LIN {X 0,Y 236.728,Z 519.016,A -85,B 0,C 180,E1 -22919.006,E2 -22919.006} C_VEL
LIN {X 0,Y 244.263,Z 527.464,A -85,B 0,C 180,E1 -22920.717,E2 -22920.717} C_VEL
LIN {X 0,Y 253.073,Z 536.486,A -85,B 0,C 180,E1 -22922.703,E2 -22922.703} C_VEL
LIN {X 0,Y 263.693,Z 545.897,A -85,B 0,C 180,E1 -22924.98,E2 -22924.98} C_VEL
LIN {X 0,Y 276.829,Z 555.997,A -85,B 0,C 180,E1 -22927.616,E2 -22927.616} C_VEL
LIN {X 0,Y 290.969,Z 566.15,A -85,B 0,C 180,E1 -22930.387,E2 -22930.387} C_VEL
LIN {X 0,Y 300.035,Z 572.76,A -85,B 0,C 180,E1 -22932.271,E2 -22932.271} C_VEL
LIN {X 0,Y 305.154,Z 576.298,A -85,B 0,C 180,E1 -22933.437,E2 -22933.437} C_VEL
LIN {X 0,Y 312.329,Z 581.44,A -85,B 0,C 180,E1 -22935.368,E2 -22935.368} C_VEL
LIN {X 0,Y 318.737,Z 585.432,A -85,B 0,C 180,E1 -22937.262,E2 -22937.262} C_VEL
LIN {X 0,Y 322.774,Z 588.128,A -85,B 0,C 180,E1 -22938.699,E2 -22938.699} C_VEL
LIN {X 0,Y 327.517,Z 591.436,A -85,B 0,C 180,E1 -22940.777,E2 -22940.777} C_VEL
LIN {X 0,Y 331.257,Z 593.607,A -85,B 0,C 180,E1 -22942.686,E2 -22942.686} C_VEL
LIN {X 0,Y 333.425,Z 594.669,A -85,B 0,C 180,E1 -22943.95,E2 -22943.95} C_VEL
LIN {X 0,Y 335.159,Z 595.455,A -85,B 0,C 180,E1 -22945.188,E2 -22945.188} C_VEL
LIN {X 0,Y 336.581,Z 595.99,A -85,B 0,C 180,E1 -22946.408,E2 -22946.408} C_VEL
LIN {X 0,Y 337.614,Z 596.404,A -85,B 0,C 180,E1 -22947.687,E2 -22947.687} C_VEL
LIN {X 0,Y 338.056,Z 596.662,A -85,B 0,C 180,E1 -22948.808,E2 -22948.808} C_VEL
LIN {X 0,Y 338.329,Z 596.679,A -85,B 0,C 180,E1 -22950,E2 -22950} C_VEL
LIN {X 0,Y 338.087,Z 596.63,A -85,B 0,C 180,E1 -22951.191,E2 -22951.191} C_VEL
LIN {X 0,Y 337.557,Z 596.361,A -85,B 0,C 180,E1 -22952.386,E2 -22952.386} C_VEL
LIN {X 0,Y 336.568,Z 595.974,A -85,B 0,C 180,E1 -22953.591,E2 -22953.591} C_VEL
LIN {X 0,Y 335.099,Z 595.465,A -85,B 0,C 180,E1 -22954.812,E2 -22954.812} C_VEL
LIN {X 0,Y 332.514,Z 594.273,A -85,B 0,C 180,E1 -22956.599,E2 -22956.599} C_VEL
LIN {X 0,Y 327.516,Z 591.416,A -85,B 0,C 180,E1 -22959.222,E2 -22959.222} C_VEL
LIN {X 0,Y 322.595,Z 587.972,A -85,B 0,C 180,E1 -22961.378,E2 -22961.378} C_VEL
LIN {X 0,Y 317.51,Z 584.709,A -85,B 0,C 180,E1 -22963.116,E2 -22963.116} C_VEL
LIN {X 0,Y 312.34,Z 581.41,A -85,B 0,C 180,E1 -22964.64,E2 -22964.64} C_VEL
LIN {X 0,Y 305.088,Z 576.303,A -85,B 0,C 180,E1 -22966.566,E2 -22966.566} C_VEL
LIN {X 0,Y 298.32,Z 571.62,A -85,B 0,C 180,E1 -22968.091,E2 -22968.091} C_VEL
LIN {X 0,Y 288.226,Z 564.238,A -85,B 0,C 180,E1 -22970.155,E2 -22970.155} C_VEL
LIN {X 0,Y 274.506,Z 554.347,A -85,B 0,C 180,E1 -22972.829,E2 -22972.829} C_VEL
LIN {X 0,Y 261.578,Z 544.164,A -85,B 0,C 180,E1 -22975.459,E2 -22975.459} C_VEL
LIN {X 0,Y 249.228,Z 532.777,A -85,B 0,C 180,E1 -22978.145,E2 -22978.145} C_VEL
LIN {X 0,Y 238.85,Z 521.493,A -85,B 0,C 180,E1 -22980.508,E2 -22980.508} C_VEL
LIN {X 0,Y 230.342,Z 511.194,A -85,B 0,C 180,E1 -22982.456,E2 -22982.456} C_VEL
LIN {X 0,Y 222.039,Z 500.025,A -85,B 0,C 180,E1 -22984.323,E2 -22984.323} C_VEL
LIN {X 0,Y 214.349,Z 487.813,A -85,B 0,C 180,E1 -22986.246,E2 -22986.246} C_VEL
LIN {X 0,Y 207.911,Z 475.576,A -85,B 0,C 180,E1 -22988.093,E2 -22988.093} C_VEL
LIN {X 0,Y 200.375,Z 459.074,A -85,B 0,C 180,E1 -22990.575,E2 -22990.575} C_VEL
LIN {X 0,Y 193.887,Z 446.712,A -85,B 0,C 180,E1 -22992.86,E2 -22992.86} C_VEL
LIN {X 0,Y 186.703,Z 434.875,A -85,B 0,C 180,E1 -22995.592,E2 -22995.592} C_VEL
LIN {X 0,Y 180.616,Z 426.163,A -85,B 0,C 180,E1 -22998.122,E2 -22998.122} C_VEL
LIN {X 0,Y 177.895,Z 422.29,A -85,B 0,C 180,E1 -22999.351,E2 -22999.351} C_VEL
LIN {X 0,Y 175.543,Z 419.17,A -85,B 0,C 180,E1 -23000.457,E2 -23000.457} C_VEL
LIN {X 0,Y 174.806,Z 417.866,A -85,B 0,C 180,E1 -23000.836,E2 -23000.836} C_VEL
LIN {X 0,Y 172.532,Z 415.661,A -85,B 0,C 180,E1 -23001.925,E2 -23001.925} C_VEL
LIN {X 0,Y 171.492,Z 413.209,A -85,B 0,C 180,E1 -23002.718,E2 -23002.718} C_VEL
LIN {X 0,Y 171.419,Z 412.642,A -85,B 0,C 180,E1 -23003.526,E2 -23003.526} C_VEL
LIN {X 0,Y 171.453,Z 412.622,A -85,B 0,C 180,E1 -23009.405,E2 -23009.405} C_VEL
LIN {X 0,Y 171.464,Z 412.598,A -85,B 0,C 180,E1 -23014.384,E2 -23014.384} C_VEL
LIN {X 0,Y 171.575,Z 412.566,A -85,B 0,C 180,E1 -23020.873,E2 -23020.873} C_VEL
LIN {X 0,Y 171.606,Z 412.607,A -85,B 0,C 180,E1 -23025.777,E2 -23025.777} C_VEL
LIN {X 0,Y 171.887,Z 412.522,A -85,B 0,C 180,E1 -23030.588,E2 -23030.588} C_VEL
LIN {X 0,Y 171.822,Z 412.58,A -85,B 0,C 180,E1 -23035.309,E2 -23035.309} C_VEL
LIN {X 0,Y 172.328,Z 412.463,A -85,B 0,C 180,E1 -23040.001,E2 -23040.001} C_VEL
LIN {X 0,Y 171.822,Z 412.582,A -85,B 0,C 180,E1 -23044.694,E2 -23044.694} C_VEL
LIN {X 0,Y 171.871,Z 412.52,A -85,B 0,C 180,E1 -23049.415,E2 -23049.415} C_VEL
LIN {X 0,Y 171.601,Z 412.606,A -85,B 0,C 180,E1 -23054.226,E2 -23054.226} C_VEL
LIN {X 0,Y 171.542,Z 412.57,A -85,B 0,C 180,E1 -23059.563,E2 -23059.563} C_VEL
LIN {X 0,Y 171.461,Z 412.589,A -85,B 0,C 180,E1 -23065.613,E2 -23065.613} C_VEL
LIN {X 0,Y 171.457,Z 412.629,A -85,B 0,C 180,E1 -23070.598,E2 -23070.598} C_VEL
LIN {X 0,Y 171.435,Z 412.785,A -85,B 0,C 180,E1 -23076.473,E2 -23076.473} C_VEL
LIN {X 0,Y 171.688,Z 413.83,A -85,B 0,C 180,E1 -23077.143,E2 -23077.143} C_VEL
LIN {X 0,Y 173.195,Z 416.474,A -85,B 0,C 180,E1 -23078.023,E2 -23078.023} C_VEL
LIN {X 0,Y 175.673,Z 419.602,A -85,B 0,C 180,E1 -23079.236,E2 -23079.236} C_VEL
LIN {X 0,Y 178.708,Z 424.182,A -85,B 0,C 180,E1 -23080.681,E2 -23080.681} C_VEL
LIN {X 0,Y 184.514,Z 434.276,A -85,B 0,C 180,E1 -23083.285,E2 -23083.285} C_VEL
LIN {X 0,Y 191.758,Z 448.084,A -85,B 0,C 180,E1 -23086.225,E2 -23086.225} C_VEL
LIN {X 0,Y 198.367,Z 463.492,A -85,B 0,C 180,E1 -23088.744,E2 -23088.744} C_VEL
LIN {X 0,Y 200.007,Z 468.221,A -85,B 0,C 180,E1 -23089.371,E2 -23089.371} C_VEL
LIN {X 0,Y 201.452,Z 479.472,A -85,B 0,C 180,E1 -23090.232,E2 -23090.232} C_VEL
LIN {X 0,Y 199.102,Z 520.445,A -85,B 0,C 180,E1 -23091.619,E2 -23091.619} C_VEL
LIN {X 0,Y 198.002,Z 530.704,A -85,B 0,C 180,E1 -23092.185,E2 -23092.185} C_VEL
LIN {X 0,Y 196.533,Z 540.028,A -85,B 0,C 180,E1 -23092.884,E2 -23092.884} C_VEL
LIN {X 0,Y 194.673,Z 549.117,A -85,B 0,C 180,E1 -23093.762,E2 -23093.762} C_VEL
LIN {X 0,Y 192.446,Z 558.257,A -85,B 0,C 180,E1 -23094.889,E2 -23094.889} C_VEL
LIN {X 0,Y 189.964,Z 567.255,A -85,B 0,C 180,E1 -23096.294,E2 -23096.294} C_VEL
LIN {X 0,Y 187.186,Z 575.977,A -85,B 0,C 180,E1 -23097.973,E2 -23097.973} C_VEL
LIN {X 0,Y 184.617,Z 583.395,A -85,B 0,C 180,E1 -23099.71,E2 -23099.71} C_VEL
LIN {X 0,Y 181.224,Z 592.186,A -85,B 0,C 180,E1 -23102.267,E2 -23102.267} C_VEL
LIN {X 0,Y 178.889,Z 598.176,A -85,B 0,C 180,E1 -23104.397,E2 -23104.397} C_VEL
LIN {X 0,Y 176.422,Z 604.491,A -85,B 0,C 180,E1 -23107.146,E2 -23107.146} C_VEL
LIN {X 0,Y 174.145,Z 609.763,A -85,B 0,C 180,E1 -23109.939,E2 -23109.939} C_VEL
LIN {X 0,Y 171.876,Z 614.855,A -85,B 0,C 180,E1 -23113.369,E2 -23113.369} C_VEL
LIN {X 0,Y 170.402,Z 618.826,A -85,B 0,C 180,E1 -23116.89,E2 -23116.89} C_VEL
LIN {X 0,Y 169.425,Z 621.766,A -85,B 0,C 180,E1 -23120.45,E2 -23120.45} C_VEL
LIN {X 0,Y 169.076,Z 623.272,A -85,B 0,C 180,E1 -23122.837,E2 -23122.837} C_VEL
LIN {X 0,Y 168.87,Z 624.806,A -85,B 0,C 180,E1 -23127.616,E2 -23127.616} C_VEL
LIN {X 0,Y 168.968,Z 625.09,A -85,B 0,C 180,E1 -23130.001,E2 -23130.001} C_VEL
LIN {X 0,Y 168.866,Z 624.204,A -85,B 0,C 180,E1 -23134.775,E2 -23134.775} C_VEL
LIN {X 0,Y 169.043,Z 623.271,A -85,B 0,C 180,E1 -23137.166,E2 -23137.166} C_VEL
LIN {X 0,Y 169.229,Z 622.38,A -85,B 0,C 180,E1 -23138.579,E2 -23138.579} C_VEL
LIN {X 0,Y 168.959,Z 621.139,A -85,B 0,C 180,E1 -23140.532,E2 -23140.532} C_VEL
LIN {X 0,Y 167.045,Z 618.534,A -85,B 0,C 180,E1 -23143.742,E2 -23143.742} C_VEL
LIN {X 0,Y 165.569,Z 615.248,A -85,B 0,C 180,E1 -23146.93,E2 -23146.93} C_VEL
LIN {X 0,Y 165.975,Z 612.775,A -85,B 0,C 180,E1 -23148.781,E2 -23148.781} C_VEL
LIN {X 0,Y 168.814,Z 606.475,A -85,B 0,C 180,E1 -23152.65,E2 -23152.65} C_VEL
LIN {X 0,Y 171.166,Z 601.299,A -85,B 0,C 180,E1 -23155.195,E2 -23155.195} C_VEL
LIN {X 0,Y 173.701,Z 595.108,A -85,B 0,C 180,E1 -23157.73,E2 -23157.73} C_VEL
LIN {X 0,Y 177.091,Z 586.895,A -85,B 0,C 180,E1 -23160.398,E2 -23160.398} C_VEL
LIN {X 0,Y 180.045,Z 579.071,A -85,B 0,C 180,E1 -23162.461,E2 -23162.461} C_VEL
LIN {X 0,Y 182.872,Z 570.992,A -85,B 0,C 180,E1 -23164.198,E2 -23164.198} C_VEL
LIN {X 0,Y 185.848,Z 561.234,A -85,B 0,C 180,E1 -23165.884,E2 -23165.884} C_VEL
LIN {X 0,Y 188.042,Z 552.846,A -85,B 0,C 180,E1 -23167.061,E2 -23167.061} C_VEL
LIN {X 0,Y 190.44,Z 542.345,A -85,B 0,C 180,E1 -23168.181,E2 -23168.181} C_VEL
LIN {X 0,Y 192.255,Z 532.052,A -85,B 0,C 180,E1 -23169.006,E2 -23169.006} C_VEL
LIN {X 0,Y 193.52,Z 521.679,A -85,B 0,C 180,E1 -23169.604,E2 -23169.604} C_VEL
LIN {X 0,Y 194.902,Z 499.84,A -85,B 0,C 180,E1 -23170.408,E2 -23170.408} C_VEL
LIN {X 0,Y 196.016,Z 479.708,A -85,B 0,C 180,E1 -23171.083,E2 -23171.083} C_VEL
LIN {X 0,Y 194.546,Z 469.953,A -85,B 0,C 180,E1 -23171.929,E2 -23171.929} C_VEL
LIN {X 0,Y 189.397,Z 457.055,A -85,B 0,C 180,E1 -23173.995,E2 -23173.995} C_VEL
LIN {X 0,Y 184.711,Z 447.009,A -85,B 0,C 180,E1 -23175.951,E2 -23175.951} C_VEL
LIN {X 0,Y 177.652,Z 433.788,A -85,B 0,C 180,E1 -23179.132,E2 -23179.132} C_VEL
LIN {X 0,Y 174.281,Z 428.326,A -85,B 0,C 180,E1 -23180.766,E2 -23180.766} C_VEL
LIN {X 0,Y 171.198,Z 423.48,A -85,B 0,C 180,E1 -23182.362,E2 -23182.362} C_VEL
LIN {X 0,Y 168.739,Z 420.14,A -85,B 0,C 180,E1 -23183.684,E2 -23183.684} C_VEL
LIN {X 0,Y 167.958,Z 418.839,A -85,B 0,C 180,E1 -23184.138,E2 -23184.138} C_VEL
LIN {X 0,Y 165.556,Z 416.617,A -85,B 0,C 180,E1 -23185.461,E2 -23185.461} C_VEL
LIN {X 0,Y 164.44,Z 414.112,A -85,B 0,C 180,E1 -23186.42,E2 -23186.42} C_VEL
LIN {X 0,Y 164.376,Z 413.526,A -85,B 0,C 180,E1 -23187.273,E2 -23187.273} C_VEL
LIN {X 0,Y 164.343,Z 413.477,A -85,B 0,C 180,E1 -23191.938,E2 -23191.938} C_VEL
LIN {X 0,Y 164.413,Z 413.469,A -85,B 0,C 180,E1 -23194.692,E2 -23194.692} C_VEL
LIN {X 0,Y 164.487,Z 413.451,A -85,B 0,C 180,E1 -23200.05,E2 -23200.05} C_VEL
LIN {X 0,Y 164.546,Z 413.477,A -85,B 0,C 180,E1 -23205.15,E2 -23205.15} C_VEL
LIN {X 0,Y 164.799,Z 413.4,A -85,B 0,C 180,E1 -23210.177,E2 -23210.177} C_VEL
LIN {X 0,Y 164.848,Z 413.407,A -85,B 0,C 180,E1 -23212.65,E2 -23212.65} C_VEL
LIN {X 0,Y 165.051,Z 413.393,A -85,B 0,C 180,E1 -23217.558,E2 -23217.558} C_VEL
LIN {X 0,Y 165.294,Z 413.339,A -85,B 0,C 180,E1 -23219.999,E2 -23219.999} C_VEL
LIN {X 0,Y 164.775,Z 413.459,A -85,B 0,C 180,E1 -23224.892,E2 -23224.892} C_VEL
LIN {X 0,Y 164.855,Z 413.419,A -85,B 0,C 180,E1 -23227.347,E2 -23227.347} C_VEL
LIN {X 0,Y 164.745,Z 413.413,A -85,B 0,C 180,E1 -23231.134,E2 -23231.134} C_VEL
LIN {X 0,Y 164.504,Z 413.456,A -85,B 0,C 180,E1 -23237.399,E2 -23237.399} C_VEL
LIN {X 0,Y 164.473,Z 413.451,A -85,B 0,C 180,E1 -23239.988,E2 -23239.988} C_VEL
LIN {X 0,Y 164.387,Z 413.474,A -85,B 0,C 180,E1 -23246.128,E2 -23246.128} C_VEL
LIN {X 0,Y 164.385,Z 413.492,A -85,B 0,C 180,E1 -23252.376,E2 -23252.376} C_VEL
LIN {X 0,Y 164.377,Z 413.826,A -85,B 0,C 180,E1 -23253.765,E2 -23253.765} C_VEL
LIN {X 0,Y 164.719,Z 415.071,A -85,B 0,C 180,E1 -23254.363,E2 -23254.363} C_VEL
LIN {X 0,Y 166.421,Z 417.681,A -85,B 0,C 180,E1 -23255.43,E2 -23255.43} C_VEL
LIN {X 0,Y 168.282,Z 419.225,A -85,B 0,C 180,E1 -23256.427,E2 -23256.427} C_VEL
LIN {X 0,Y 170.447,Z 422.668,A -85,B 0,C 180,E1 -23257.643,E2 -23257.643} C_VEL
LIN {X 0,Y 172.045,Z 424.419,A -85,B 0,C 180,E1 -23258.448,E2 -23258.448} C_VEL
LIN {X 0,Y 174.727,Z 428.084,A -85,B 0,C 180,E1 -23259.782,E2 -23259.782} C_VEL
LIN {X 0,Y 181.199,Z 437.59,A -85,B 0,C 180,E1 -23262.745,E2 -23262.745} C_VEL
LIN {X 0,Y 186.924,Z 446.683,A -85,B 0,C 180,E1 -23265.11,E2 -23265.11} C_VEL
LIN {X 0,Y 192.646,Z 456.992,A -85,B 0,C 180,E1 -23267.308,E2 -23267.308} C_VEL
LIN {X 0,Y 199.199,Z 470.707,A -85,B 0,C 180,E1 -23269.675,E2 -23269.675} C_VEL
LIN {X 0,Y 206.608,Z 486.849,A -85,B 0,C 180,E1 -23272.111,E2 -23272.111} C_VEL
LIN {X 0,Y 215.246,Z 501.527,A -85,B 0,C 180,E1 -23274.484,E2 -23274.484} C_VEL
LIN {X 0,Y 223.669,Z 513.611,A -85,B 0,C 180,E1 -23276.575,E2 -23276.575} C_VEL
LIN {X 0,Y 233.428,Z 525.815,A -85,B 0,C 180,E1 -23279.036,E2 -23279.036} C_VEL
LIN {X 0,Y 242.728,Z 536.201,A -85,B 0,C 180,E1 -23281.369,E2 -23281.369} C_VEL
LIN {X 0,Y 253.999,Z 546.99,A -85,B 0,C 180,E1 -23284.058,E2 -23284.058} C_VEL
LIN {X 0,Y 267.274,Z 557.559,A -85,B 0,C 180,E1 -23286.971,E2 -23286.971} C_VEL
LIN {X 0,Y 280.838,Z 567.195,A -85,B 0,C 180,E1 -23289.787,E2 -23289.787} C_VEL
LIN {X 0,Y 289.684,Z 573.411,A -85,B 0,C 180,E1 -23291.615,E2 -23291.615} C_VEL
LIN {X 0,Y 298.819,Z 579.758,A -85,B 0,C 180,E1 -23293.606,E2 -23293.606} C_VEL
LIN {X 0,Y 305.423,Z 584.503,A -85,B 0,C 180,E1 -23295.338,E2 -23295.338} C_VEL
LIN {X 0,Y 311.033,Z 588.132,A -85,B 0,C 180,E1 -23296.941,E2 -23296.941} C_VEL
LIN {X 0,Y 315.717,Z 591.005,A -85,B 0,C 180,E1 -23298.443,E2 -23298.443} C_VEL
LIN {X 0,Y 320.624,Z 594.537,A -85,B 0,C 180,E1 -23300.53,E2 -23300.53} C_VEL
LIN {X 0,Y 324.704,Z 597.007,A -85,B 0,C 180,E1 -23302.538,E2 -23302.538} C_VEL
LIN {X 0,Y 327,Z 598.172,A -85,B 0,C 180,E1 -23303.831,E2 -23303.831} C_VEL
LIN {X 0,Y 328.877,Z 599.073,A -85,B 0,C 180,E1 -23305.096,E2 -23305.096} C_VEL
LIN {X 0,Y 330.825,Z 599.849,A -85,B 0,C 180,E1 -23306.805,E2 -23306.805} C_VEL
LIN {X 0,Y 331.432,Z 600.068,A -85,B 0,C 180,E1 -23307.569,E2 -23307.569} C_VEL
LIN {X 0,Y 331.976,Z 600.353,A -85,B 0,C 180,E1 -23308.787,E2 -23308.787} C_VEL
LIN {X 0,Y 332.28,Z 600.374,A -85,B 0,C 180,E1 -23310,E2 -23310} C_VEL
LIN {X 0,Y 332.008,Z 600.326,A -85,B 0,C 180,E1 -23311.213,E2 -23311.213} C_VEL
LIN {X 0,Y 330.825,Z 599.859,A -85,B 0,C 180,E1 -23313.194,E2 -23313.194} C_VEL
LIN {X 0,Y 328.815,Z 599.085,A -85,B 0,C 180,E1 -23314.904,E2 -23314.904} C_VEL
LIN {X 0,Y 325.669,Z 597.531,A -85,B 0,C 180,E1 -23316.939,E2 -23316.939} C_VEL
LIN {X 0,Y 322.095,Z 595.476,A -85,B 0,C 180,E1 -23318.785,E2 -23318.785} C_VEL
LIN {X 0,Y 319.133,Z 593.487,A -85,B 0,C 180,E1 -23320.147,E2 -23320.147} C_VEL
LIN {X 0,Y 315.653,Z 590.975,A -85,B 0,C 180,E1 -23321.581,E2 -23321.581} C_VEL
LIN {X 0,Y 310.442,Z 587.771,A -85,B 0,C 180,E1 -23323.233,E2 -23323.233} C_VEL
LIN {X 0,Y 305.203,Z 584.349,A -85,B 0,C 180,E1 -23324.731,E2 -23324.731} C_VEL
LIN {X 0,Y 298.782,Z 579.747,A -85,B 0,C 180,E1 -23326.395,E2 -23326.395} C_VEL
LIN {X 0,Y 289.661,Z 573.417,A -85,B 0,C 180,E1 -23328.385,E2 -23328.385} C_VEL
LIN {X 0,Y 278.12,Z 565.341,A -85,B 0,C 180,E1 -23330.778,E2 -23330.778} C_VEL
LIN {X 0,Y 263.246,Z 554.562,A -85,B 0,C 180,E1 -23333.883,E2 -23333.883} C_VEL
LIN {X 0,Y 251.277,Z 544.483,A -85,B 0,C 180,E1 -23336.583,E2 -23336.583} C_VEL
LIN {X 0,Y 241.139,Z 534.456,A -85,B 0,C 180,E1 -23339.034,E2 -23339.034} C_VEL
LIN {X 0,Y 231.156,Z 523.114,A -85,B 0,C 180,E1 -23341.534,E2 -23341.534} C_VEL
LIN {X 0,Y 222.069,Z 511.424,A -85,B 0,C 180,E1 -23343.826,E2 -23343.826} C_VEL
LIN {X 0,Y 212.518,Z 497.302,A -85,B 0,C 180,E1 -23346.22,E2 -23346.22} C_VEL
LIN {X 0,Y 204.497,Z 482.639,A -85,B 0,C 180,E1 -23348.54,E2 -23348.54} C_VEL
LIN {X 0,Y 195.455,Z 462.655,A -85,B 0,C 180,E1 -23351.657,E2 -23351.657} C_VEL
LIN {X 0,Y 189.424,Z 450.986,A -85,B 0,C 180,E1 -23353.914,E2 -23353.914} C_VEL
LIN {X 0,Y 182.648,Z 439.754,A -85,B 0,C 180,E1 -23356.64,E2 -23356.64} C_VEL
LIN {X 0,Y 177.085,Z 431.544,A -85,B 0,C 180,E1 -23359.093,E2 -23359.093} C_VEL
LIN {X 0,Y 174.236,Z 427.557,A -85,B 0,C 180,E1 -23360.447,E2 -23360.447} C_VEL
LIN {X 0,Y 171.306,Z 423.48,A -85,B 0,C 180,E1 -23361.929,E2 -23361.929} C_VEL
LIN {X 0,Y 169.048,Z 420.726,A -85,B 0,C 180,E1 -23363.116,E2 -23363.116} C_VEL
LIN {X 0,Y 167.933,Z 418.825,A -85,B 0,C 180,E1 -23363.764,E2 -23363.764} C_VEL
LIN {X 0,Y 165.584,Z 416.669,A -85,B 0,C 180,E1 -23365.057,E2 -23365.057} C_VEL
LIN {X 0,Y 164.44,Z 414.038,A -85,B 0,C 180,E1 -23366.041,E2 -23366.041} C_VEL
LIN {X 0,Y 164.345,Z 413.513,A -85,B 0,C 180,E1 -23366.923,E2 -23366.923} C_VEL
LIN {X 0,Y 164.401,Z 413.504,A -85,B 0,C 180,E1 -23369.138,E2 -23369.138} C_VEL
LIN {X 0,Y 164.412,Z 413.479,A -85,B 0,C 180,E1 -23374.695,E2 -23374.695} C_VEL
LIN {X 0,Y 164.48,Z 413.45,A -85,B 0,C 180,E1 -23380.052,E2 -23380.052} C_VEL
LIN {X 0,Y 164.549,Z 413.489,A -85,B 0,C 180,E1 -23385.153,E2 -23385.153} C_VEL
LIN {X 0,Y 164.801,Z 413.402,A -85,B 0,C 180,E1 -23390.18,E2 -23390.18} C_VEL
LIN {X 0,Y 164.851,Z 413.419,A -85,B 0,C 180,E1 -23392.653,E2 -23392.653} C_VEL
LIN {X 0,Y 165.047,Z 413.382,A -85,B 0,C 180,E1 -23397.561,E2 -23397.561} C_VEL
LIN {X 0,Y 165.291,Z 413.339,A -85,B 0,C 180,E1 -23400.001,E2 -23400.001} C_VEL
LIN {X 0,Y 164.771,Z 413.46,A -85,B 0,C 180,E1 -23404.895,E2 -23404.895} C_VEL
LIN {X 0,Y 164.844,Z 413.408,A -85,B 0,C 180,E1 -23407.35,E2 -23407.35} C_VEL
LIN {X 0,Y 164.748,Z 413.416,A -85,B 0,C 180,E1 -23411.148,E2 -23411.148} C_VEL
LIN {X 0,Y 164.49,Z 413.447,A -85,B 0,C 180,E1 -23417.404,E2 -23417.404} C_VEL
LIN {X 0,Y 164.472,Z 413.453,A -85,B 0,C 180,E1 -23419.991,E2 -23419.991} C_VEL
LIN {X 0,Y 164.387,Z 413.467,A -85,B 0,C 180,E1 -23426.132,E2 -23426.132} C_VEL
LIN {X 0,Y 164.388,Z 413.505,A -85,B 0,C 180,E1 -23432.38,E2 -23432.38} C_VEL
LIN {X 0,Y 164.388,Z 413.886,A -85,B 0,C 180,E1 -23433.418,E2 -23433.418} C_VEL
LIN {X 0,Y 164.851,Z 415.357,A -85,B 0,C 180,E1 -23434.077,E2 -23434.077} C_VEL
LIN {X 0,Y 166.518,Z 417.759,A -85,B 0,C 180,E1 -23435.097,E2 -23435.097} C_VEL
LIN {X 0,Y 168.305,Z 419.258,A -85,B 0,C 180,E1 -23436.054,E2 -23436.054} C_VEL
LIN {X 0,Y 170.355,Z 422.505,A -85,B 0,C 180,E1 -23437.205,E2 -23437.205} C_VEL
LIN {X 0,Y 172.352,Z 425.179,A -85,B 0,C 180,E1 -23438.241,E2 -23438.241} C_VEL
LIN {X 0,Y 176.255,Z 431.544,A -85,B 0,C 180,E1 -23440.206,E2 -23440.206} C_VEL
LIN {X 0,Y 180.512,Z 439.006,A -85,B 0,C 180,E1 -23442.202,E2 -23442.202} C_VEL
LIN {X 0,Y 187.332,Z 452.339,A -85,B 0,C 180,E1 -23445.148,E2 -23445.148} C_VEL
LIN {X 0,Y 194.157,Z 468.716,A -85,B 0,C 180,E1 -23447.908,E2 -23447.908} C_VEL
LIN {X 0,Y 194.9,Z 471.646,A -85,B 0,C 180,E1 -23448.245,E2 -23448.245} C_VEL
LIN {X 0,Y 195.961,Z 480.953,A -85,B 0,C 180,E1 -23448.963,E2 -23448.963} C_VEL
LIN {X 0,Y 193.606,Z 520.134,A -85,B 0,C 180,E1 -23450.311,E2 -23450.311} C_VEL
LIN {X 0,Y 192.382,Z 530.958,A -85,B 0,C 180,E1 -23450.918,E2 -23450.918} C_VEL
LIN {X 0,Y 190.676,Z 541.095,A -85,B 0,C 180,E1 -23451.709,E2 -23451.709} C_VEL
LIN {X 0,Y 188.532,Z 550.889,A -85,B 0,C 180,E1 -23452.718,E2 -23452.718} C_VEL
LIN {X 0,Y 186.248,Z 559.651,A -85,B 0,C 180,E1 -23453.873,E2 -23453.873} C_VEL
LIN {X 0,Y 183.674,Z 568.372,A -85,B 0,C 180,E1 -23455.309,E2 -23455.309} C_VEL
LIN {X 0,Y 180.799,Z 576.879,A -85,B 0,C 180,E1 -23457.031,E2 -23457.031} C_VEL
LIN {X 0,Y 178.49,Z 583.199,A -85,B 0,C 180,E1 -23458.554,E2 -23458.554} C_VEL
LIN {X 0,Y 174.946,Z 591.99,A -85,B 0,C 180,E1 -23461.181,E2 -23461.181} C_VEL
LIN {X 0,Y 172.483,Z 597.98,A -85,B 0,C 180,E1 -23463.372,E2 -23463.372} C_VEL
LIN {X 0,Y 169.872,Z 604.295,A -85,B 0,C 180,E1 -23466.211,E2 -23466.211} C_VEL
LIN {X 0,Y 167.452,Z 609.567,A -85,B 0,C 180,E1 -23469.1,E2 -23469.1} C_VEL
LIN {X 0,Y 165.068,Z 614.66,A -85,B 0,C 180,E1 -23472.661,E2 -23472.661} C_VEL
LIN {X 0,Y 163.452,Z 618.629,A -85,B 0,C 180,E1 -23476.322,E2 -23476.322} C_VEL
LIN {X 0,Y 162.405,Z 621.571,A -85,B 0,C 180,E1 -23480.033,E2 -23480.033} C_VEL
LIN {X 0,Y 162.002,Z 623.076,A -85,B 0,C 180,E1 -23482.523,E2 -23482.523} C_VEL
LIN {X 0,Y 161.8,Z 624.612,A -85,B 0,C 180,E1 -23487.511,E2 -23487.511} C_VEL
LIN {X 0,Y 161.884,Z 624.895,A -85,B 0,C 180,E1 -23490.001,E2 -23490.001} C_VEL
LIN {X 0,Y 161.771,Z 624.009,A -85,B 0,C 180,E1 -23494.985,E2 -23494.985} C_VEL
LIN {X 0,Y 162.149,Z 622.327,A -85,B 0,C 180,E1 -23498.719,E2 -23498.719} C_VEL
LIN {X 0,Y 163.452,Z 618.628,A -85,B 0,C 180,E1 -23503.68,E2 -23503.68} C_VEL
LIN {X 0,Y 165.063,Z 614.658,A -85,B 0,C 180,E1 -23507.341,E2 -23507.341} C_VEL
LIN {X 0,Y 165.975,Z 612.775,A -85,B 0,C 180,E1 -23508.781,E2 -23508.781} C_VEL
LIN {X 0,Y 166.522,Z 610.192,A -85,B 0,C 180,E1 -23510.581,E2 -23510.581} C_VEL
LIN {X 0,Y 165.941,Z 605.51,A -85,B 0,C 180,E1 -23513.589,E2 -23513.589} C_VEL
LIN {X 0,Y 165.656,Z 600.32,A -85,B 0,C 180,E1 -23516.524,E2 -23516.524} C_VEL
LIN {X 0,Y 166.652,Z 596.784,A -85,B 0,C 180,E1 -23518.148,E2 -23518.148} C_VEL
LIN {X 0,Y 170.23,Z 588.548,A -85,B 0,C 180,E1 -23521.069,E2 -23521.069} C_VEL
LIN {X 0,Y 174.084,Z 578.875,A -85,B 0,C 180,E1 -23523.718,E2 -23523.718} C_VEL
LIN {X 0,Y 177.046,Z 570.797,A -85,B 0,C 180,E1 -23525.49,E2 -23525.49} C_VEL
LIN {X 0,Y 180.134,Z 561.039,A -85,B 0,C 180,E1 -23527.21,E2 -23527.21} C_VEL
LIN {X 0,Y 182.441,Z 552.651,A -85,B 0,C 180,E1 -23528.402,E2 -23528.402} C_VEL
LIN {X 0,Y 184.919,Z 542.151,A -85,B 0,C 180,E1 -23529.539,E2 -23529.539} C_VEL
LIN {X 0,Y 186.827,Z 531.734,A -85,B 0,C 180,E1 -23530.38,E2 -23530.38} C_VEL
LIN {X 0,Y 188.082,Z 521.544,A -85,B 0,C 180,E1 -23530.985,E2 -23530.985} C_VEL
LIN {X 0,Y 189.541,Z 499.766,A -85,B 0,C 180,E1 -23531.797,E2 -23531.797} C_VEL
LIN {X 0,Y 190.654,Z 480.823,A -85,B 0,C 180,E1 -23532.437,E2 -23532.437} C_VEL
LIN {X 0,Y 189.402,Z 472.537,A -85,B 0,C 180,E1 -23533.202,E2 -23533.202} C_VEL
LIN {X 0,Y 184.087,Z 459.259,A -85,B 0,C 180,E1 -23535.482,E2 -23535.482} C_VEL
LIN {X 0,Y 180.111,Z 450.731,A -85,B 0,C 180,E1 -23537.261,E2 -23537.261} C_VEL
LIN {X 0,Y 173.86,Z 438.725,A -85,B 0,C 180,E1 -23540.275,E2 -23540.275} C_VEL
LIN {X 0,Y 170.411,Z 432.987,A -85,B 0,C 180,E1 -23542.064,E2 -23542.064} C_VEL
LIN {X 0,Y 167.99,Z 429.046,A -85,B 0,C 180,E1 -23543.403,E2 -23543.403} C_VEL
LIN {X 0,Y 165.336,Z 425.183,A -85,B 0,C 180,E1 -23544.935,E2 -23544.935} C_VEL
LIN {X 0,Y 162.486,Z 422.107,A -85,B 0,C 180,E1 -23546.623,E2 -23546.623} C_VEL
LIN {X 0,Y 161.16,Z 419.831,A -85,B 0,C 180,E1 -23547.523,E2 -23547.523} C_VEL
LIN {X 0,Y 158.833,Z 417.904,A -85,B 0,C 180,E1 -23549.021,E2 -23549.021} C_VEL
LIN {X 0,Y 157.408,Z 414.944,A -85,B 0,C 180,E1 -23550.4,E2 -23550.4} C_VEL
LIN {X 0,Y 157.299,Z 414.413,A -85,B 0,C 180,E1 -23551.294,E2 -23551.294} C_VEL
LIN {X 0,Y 157.313,Z 414.373,A -85,B 0,C 180,E1 -23556.29,E2 -23556.29} C_VEL
LIN {X 0,Y 157.417,Z 414.324,A -85,B 0,C 180,E1 -23561.787,E2 -23561.787} C_VEL
LIN {X 0,Y 157.552,Z 414.338,A -85,B 0,C 180,E1 -23567.111,E2 -23567.111} C_VEL
LIN {X 0,Y 157.728,Z 414.282,A -85,B 0,C 180,E1 -23569.732,E2 -23569.732} C_VEL
LIN {X 0,Y 157.805,Z 414.279,A -85,B 0,C 180,E1 -23572.32,E2 -23572.32} C_VEL
LIN {X 0,Y 158.257,Z 414.214,A -85,B 0,C 180,E1 -23579.999,E2 -23579.999} C_VEL
LIN {X 0,Y 157.811,Z 414.289,A -85,B 0,C 180,E1 -23587.676,E2 -23587.676} C_VEL
LIN {X 0,Y 157.676,Z 414.293,A -85,B 0,C 180,E1 -23591.306,E2 -23591.306} C_VEL
LIN {X 0,Y 157.478,Z 414.36,A -85,B 0,C 180,E1 -23595.53,E2 -23595.53} C_VEL
LIN {X 0,Y 157.369,Z 414.342,A -85,B 0,C 180,E1 -23600.931,E2 -23600.931} C_VEL
LIN {X 0,Y 157.308,Z 414.351,A -85,B 0,C 180,E1 -23606.679,E2 -23606.679} C_VEL
LIN {X 0,Y 157.339,Z 414.676,A -85,B 0,C 180,E1 -23609.703,E2 -23609.703} C_VEL
LIN {X 0,Y 157.689,Z 415.857,A -85,B 0,C 180,E1 -23610.46,E2 -23610.46} C_VEL
LIN {X 0,Y 159.215,Z 418.377,A -85,B 0,C 180,E1 -23611.632,E2 -23611.632} C_VEL
LIN {X 0,Y 161.46,Z 420.154,A -85,B 0,C 180,E1 -23613.054,E2 -23613.054} C_VEL
LIN {X 0,Y 163.49,Z 423.459,A -85,B 0,C 180,E1 -23614.394,E2 -23614.394} C_VEL
LIN {X 0,Y 165.522,Z 425.569,A -85,B 0,C 180,E1 -23615.571,E2 -23615.571} C_VEL
LIN {X 0,Y 167.969,Z 429.04,A -85,B 0,C 180,E1 -23616.973,E2 -23616.973} C_VEL
LIN {X 0,Y 169.204,Z 430.642,A -85,B 0,C 180,E1 -23617.639,E2 -23617.639} C_VEL
LIN {X 0,Y 175.22,Z 439.293,A -85,B 0,C 180,E1 -23620.675,E2 -23620.675} C_VEL
LIN {X 0,Y 181.544,Z 449.222,A -85,B 0,C 180,E1 -23623.524,E2 -23623.524} C_VEL
LIN {X 0,Y 187.875,Z 460.689,A -85,B 0,C 180,E1 -23626.135,E2 -23626.135} C_VEL
LIN {X 0,Y 193.898,Z 473.486,A -85,B 0,C 180,E1 -23628.458,E2 -23628.458} C_VEL
LIN {X 0,Y 201.993,Z 491.356,A -85,B 0,C 180,E1 -23631.279,E2 -23631.279} C_VEL
LIN {X 0,Y 210.523,Z 506.075,A -85,B 0,C 180,E1 -23633.746,E2 -23633.746} C_VEL
LIN {X 0,Y 218.434,Z 517.873,A -85,B 0,C 180,E1 -23635.942,E2 -23635.942} C_VEL
LIN {X 0,Y 227.023,Z 529.009,A -85,B 0,C 180,E1 -23638.352,E2 -23638.352} C_VEL
LIN {X 0,Y 234.425,Z 537.612,A -85,B 0,C 180,E1 -23640.388,E2 -23640.388} C_VEL
LIN {X 0,Y 244.429,Z 547.815,A -85,B 0,C 180,E1 -23643.039,E2 -23643.039} C_VEL
LIN {X 0,Y 254.755,Z 556.641,A -85,B 0,C 180,E1 -23645.555,E2 -23645.555} C_VEL
LIN {X 0,Y 269.098,Z 567.114,A -85,B 0,C 180,E1 -23648.778,E2 -23648.778} C_VEL
LIN {X 0,Y 281.65,Z 575.581,A -85,B 0,C 180,E1 -23651.477,E2 -23651.477} C_VEL
LIN {X 0,Y 292.579,Z 582.992,A -85,B 0,C 180,E1 -23653.908,E2 -23653.908} C_VEL
LIN {X 0,Y 299.527,Z 587.974,A -85,B 0,C 180,E1 -23655.705,E2 -23655.705} C_VEL
LIN {X 0,Y 304.737,Z 591.358,A -85,B 0,C 180,E1 -23657.167,E2 -23657.167} C_VEL
LIN {X 0,Y 309.786,Z 594.475,A -85,B 0,C 180,E1 -23658.77,E2 -23658.77} C_VEL
LIN {X 0,Y 315.026,Z 598.177,A -85,B 0,C 180,E1 -23661.015,E2 -23661.015} C_VEL
LIN {X 0,Y 318.736,Z 600.427,A -85,B 0,C 180,E1 -23662.847,E2 -23662.847} C_VEL
LIN {X 0,Y 322.233,Z 602.162,A -85,B 0,C 180,E1 -23664.995,E2 -23664.995} C_VEL
LIN {X 0,Y 323.946,Z 602.89,A -85,B 0,C 180,E1 -23666.334,E2 -23666.334} C_VEL
LIN {X 0,Y 325.059,Z 603.308,A -85,B 0,C 180,E1 -23667.521,E2 -23667.521} C_VEL
LIN {X 0,Y 325.655,Z 603.606,A -85,B 0,C 180,E1 -23668.763,E2 -23668.763} C_VEL
LIN {X 0,Y 325.97,Z 603.643,A -85,B 0,C 180,E1 -23670,E2 -23670} C_VEL
LIN {X 0,Y 325.678,Z 603.588,A -85,B 0,C 180,E1 -23671.236,E2 -23671.236} C_VEL
LIN {X 0,Y 325.059,Z 603.298,A -85,B 0,C 180,E1 -23672.478,E2 -23672.478} C_VEL
LIN {X 0,Y 323.85,Z 602.851,A -85,B 0,C 180,E1 -23673.732,E2 -23673.732} C_VEL
LIN {X 0,Y 322.2,Z 602.171,A -85,B 0,C 180,E1 -23675.005,E2 -23675.005} C_VEL
LIN {X 0,Y 320.222,Z 601.202,A -85,B 0,C 180,E1 -23676.3,E2 -23676.3} C_VEL
LIN {X 0,Y 317.783,Z 599.904,A -85,B 0,C 180,E1 -23677.625,E2 -23677.625} C_VEL
LIN {X 0,Y 313.631,Z 597.242,A -85,B 0,C 180,E1 -23679.613,E2 -23679.613} C_VEL
LIN {X 0,Y 309.784,Z 594.458,A -85,B 0,C 180,E1 -23681.229,E2 -23681.229} C_VEL
LIN {X 0,Y 304.734,Z 591.384,A -85,B 0,C 180,E1 -23682.83,E2 -23682.83} C_VEL
LIN {X 0,Y 297.951,Z 586.837,A -85,B 0,C 180,E1 -23684.742,E2 -23684.742} C_VEL
LIN {X 0,Y 292.574,Z 583.008,A -85,B 0,C 180,E1 -23686.088,E2 -23686.088} C_VEL
LIN {X 0,Y 281.641,Z 575.61,A -85,B 0,C 180,E1 -23688.518,E2 -23688.518} C_VEL
LIN {X 0,Y 267.45,Z 565.985,A -85,B 0,C 180,E1 -23691.585,E2 -23691.585} C_VEL
LIN {X 0,Y 253.442,Z 555.619,A -85,B 0,C 180,E1 -23694.75,E2 -23694.75} C_VEL
LIN {X 0,Y 241.263,Z 544.795,A -85,B 0,C 180,E1 -23697.779,E2 -23697.779} C_VEL
LIN {X 0,Y 230.745,Z 533.491,A -85,B 0,C 180,E1 -23700.613,E2 -23700.613} C_VEL
LIN {X 0,Y 221.966,Z 522.576,A -85,B 0,C 180,E1 -23703.066,E2 -23703.066} C_VEL
LIN {X 0,Y 214.582,Z 512.309,A -85,B 0,C 180,E1 -23705.139,E2 -23705.139} C_VEL
LIN {X 0,Y 205.92,Z 498.513,A -85,B 0,C 180,E1 -23707.534,E2 -23707.534} C_VEL
LIN {X 0,Y 199.124,Z 485.472,A -85,B 0,C 180,E1 -23709.66,E2 -23709.66} C_VEL
LIN {X 0,Y 190.831,Z 466.717,A -85,B 0,C 180,E1 -23712.709,E2 -23712.709} C_VEL
LIN {X 0,Y 184.918,Z 455.087,A -85,B 0,C 180,E1 -23715.061,E2 -23715.061} C_VEL
LIN {X 0,Y 178.882,Z 444.895,A -85,B 0,C 180,E1 -23717.64,E2 -23717.64} C_VEL
LIN {X 0,Y 173.249,Z 436.424,A -85,B 0,C 180,E1 -23720.277,E2 -23720.277} C_VEL
LIN {X 0,Y 170.439,Z 432.474,A -85,B 0,C 180,E1 -23721.7,E2 -23721.7} C_VEL
LIN {X 0,Y 168.09,Z 429.142,A -85,B 0,C 180,E1 -23722.964,E2 -23722.964} C_VEL
LIN {X 0,Y 165.523,Z 425.593,A -85,B 0,C 180,E1 -23724.427,E2 -23724.427} C_VEL
LIN {X 0,Y 162.258,Z 421.734,A -85,B 0,C 180,E1 -23726.387,E2 -23726.387} C_VEL
LIN {X 0,Y 161.136,Z 419.835,A -85,B 0,C 180,E1 -23727.15,E2 -23727.15} C_VEL
LIN {X 0,Y 158.729,Z 417.774,A -85,B 0,C 180,E1 -23728.708,E2 -23728.708} C_VEL
LIN {X 0,Y 157.461,Z 415.141,A -85,B 0,C 180,E1 -23729.861,E2 -23729.861} C_VEL
LIN {X 0,Y 157.279,Z 414.435,A -85,B 0,C 180,E1 -23730.927,E2 -23730.927} C_VEL
LIN {X 0,Y 157.317,Z 414.351,A -85,B 0,C 180,E1 -23733.467,E2 -23733.467} C_VEL
LIN {X 0,Y 157.389,Z 414.335,A -85,B 0,C 180,E1 -23739.669,E2 -23739.669} C_VEL
LIN {X 0,Y 157.474,Z 414.361,A -85,B 0,C 180,E1 -23744.469,E2 -23744.469} C_VEL
LIN {X 0,Y 157.725,Z 414.283,A -85,B 0,C 180,E1 -23749.735,E2 -23749.735} C_VEL
LIN {X 0,Y 157.807,Z 414.289,A -85,B 0,C 180,E1 -23752.323,E2 -23752.323} C_VEL
LIN {X 0,Y 158.253,Z 414.215,A -85,B 0,C 180,E1 -23760.001,E2 -23760.001} C_VEL
LIN {X 0,Y 157.801,Z 414.28,A -85,B 0,C 180,E1 -23767.68,E2 -23767.68} C_VEL
LIN {X 0,Y 157.678,Z 414.297,A -85,B 0,C 180,E1 -23771.317,E2 -23771.317} C_VEL
LIN {X 0,Y 157.467,Z 414.343,A -85,B 0,C 180,E1 -23775.534,E2 -23775.534} C_VEL
LIN {X 0,Y 157.368,Z 414.348,A -85,B 0,C 180,E1 -23780.935,E2 -23780.935} C_VEL
LIN {X 0,Y 157.309,Z 414.347,A -85,B 0,C 180,E1 -23786.683,E2 -23786.683} C_VEL
LIN {X 0,Y 157.324,Z 414.618,A -85,B 0,C 180,E1 -23789.25,E2 -23789.25} C_VEL
LIN {X 0,Y 157.548,Z 415.519,A -85,B 0,C 180,E1 -23789.939,E2 -23789.939} C_VEL
LIN {X 0,Y 159.048,Z 418.151,A -85,B 0,C 180,E1 -23791.127,E2 -23791.127} C_VEL
LIN {X 0,Y 161.578,Z 420.399,A -85,B 0,C 180,E1 -23792.752,E2 -23792.752} C_VEL
LIN {X 0,Y 163.58,Z 423.553,A -85,B 0,C 180,E1 -23794.061,E2 -23794.061} C_VEL
LIN {X 0,Y 165.515,Z 425.555,A -85,B 0,C 180,E1 -23795.18,E2 -23795.18} C_VEL
LIN {X 0,Y 169.14,Z 430.833,A -85,B 0,C 180,E1 -23797.237,E2 -23797.237} C_VEL
LIN {X 0,Y 172.94,Z 437.18,A -85,B 0,C 180,E1 -23799.26,E2 -23799.26} C_VEL
LIN {X 0,Y 177.988,Z 446.557,A -85,B 0,C 180,E1 -23801.753,E2 -23801.753} C_VEL
LIN {X 0,Y 183.31,Z 457.387,A -85,B 0,C 180,E1 -23804.17,E2 -23804.17} C_VEL
LIN {X 0,Y 189.412,Z 472.432,A -85,B 0,C 180,E1 -23806.796,E2 -23806.796} C_VEL
LIN {X 0,Y 190.612,Z 480.939,A -85,B 0,C 180,E1 -23807.557,E2 -23807.557} C_VEL
LIN {X 0,Y 188.194,Z 519.946,A -85,B 0,C 180,E1 -23808.929,E2 -23808.929} C_VEL
LIN {X 0,Y 186.938,Z 530.713,A -85,B 0,C 180,E1 -23809.544,E2 -23809.544} C_VEL
LIN {X 0,Y 185.17,Z 540.901,A -85,B 0,C 180,E1 -23810.351,E2 -23810.351} C_VEL
LIN {X 0,Y 182.947,Z 550.694,A -85,B 0,C 180,E1 -23811.374,E2 -23811.374} C_VEL
LIN {X 0,Y 180.553,Z 559.456,A -85,B 0,C 180,E1 -23812.542,E2 -23812.542} C_VEL
LIN {X 0,Y 177.877,Z 568.177,A -85,B 0,C 180,E1 -23814.006,E2 -23814.006} C_VEL
LIN {X 0,Y 174.887,Z 576.684,A -85,B 0,C 180,E1 -23815.765,E2 -23815.765} C_VEL
LIN {X 0,Y 172.441,Z 583.003,A -85,B 0,C 180,E1 -23817.317,E2 -23817.317} C_VEL
LIN {X 0,Y 168.75,Z 591.795,A -85,B 0,C 180,E1 -23820.017,E2 -23820.017} C_VEL
LIN {X 0,Y 165.687,Z 598.787,A -85,B 0,C 180,E1 -23822.712,E2 -23822.712} C_VEL
LIN {X 0,Y 163.364,Z 604.099,A -85,B 0,C 180,E1 -23825.201,E2 -23825.201} C_VEL
LIN {X 0,Y 160.789,Z 609.371,A -85,B 0,C 180,E1 -23828.191,E2 -23828.191} C_VEL
LIN {X 0,Y 158.293,Z 614.464,A -85,B 0,C 180,E1 -23831.894,E2 -23831.894} C_VEL
LIN {X 0,Y 156.527,Z 618.433,A -85,B 0,C 180,E1 -23835.704,E2 -23835.704} C_VEL
LIN {X 0,Y 155.406,Z 621.375,A -85,B 0,C 180,E1 -23839.579,E2 -23839.579} C_VEL
LIN {X 0,Y 154.952,Z 622.881,A -85,B 0,C 180,E1 -23842.18,E2 -23842.18} C_VEL
LIN {X 0,Y 154.702,Z 624.417,A -85,B 0,C 180,E1 -23847.397,E2 -23847.397} C_VEL
LIN {X 0,Y 154.797,Z 624.701,A -85,B 0,C 180,E1 -23850.001,E2 -23850.001} C_VEL
LIN {X 0,Y 154.698,Z 623.814,A -85,B 0,C 180,E1 -23855.214,E2 -23855.214} C_VEL
LIN {X 0,Y 154.932,Z 622.88,A -85,B 0,C 180,E1 -23857.822,E2 -23857.822} C_VEL
LIN {X 0,Y 156.083,Z 619.523,A -85,B 0,C 180,E1 -23863.012,E2 -23863.012} C_VEL
LIN {X 0,Y 157.606,Z 615.891,A -85,B 0,C 180,E1 -23866.849,E2 -23866.849} C_VEL
LIN {X 0,Y 159.926,Z 611.159,A -85,B 0,C 180,E1 -23870.583,E2 -23870.583} C_VEL
LIN {X 0,Y 162.843,Z 605.189,A -85,B 0,C 180,E1 -23874.205,E2 -23874.205} C_VEL
LIN {X 0,Y 165.59,Z 599.095,A -85,B 0,C 180,E1 -23877.146,E2 -23877.146} C_VEL
LIN {X 0,Y 166.652,Z 596.784,A -85,B 0,C 180,E1 -23878.148,E2 -23878.148} C_VEL
LIN {X 0,Y 167.709,Z 593.117,A -85,B 0,C 180,E1 -23879.697,E2 -23879.697} C_VEL
LIN {X 0,Y 167.915,Z 586.689,A -85,B 0,C 180,E1 -23882.279,E2 -23882.279} C_VEL
LIN {X 0,Y 168.3,Z 579.821,A -85,B 0,C 180,E1 -23884.678,E2 -23884.678} C_VEL
LIN {X 0,Y 169.589,Z 575.205,A -85,B 0,C 180,E1 -23885.889,E2 -23885.889} C_VEL
LIN {X 0,Y 173.598,Z 563.988,A -85,B 0,C 180,E1 -23888.126,E2 -23888.126} C_VEL
LIN {X 0,Y 176.935,Z 552.456,A -85,B 0,C 180,E1 -23889.829,E2 -23889.829} C_VEL
LIN {X 0,Y 179.503,Z 541.956,A -85,B 0,C 180,E1 -23890.981,E2 -23890.981} C_VEL
LIN {X 0,Y 181.425,Z 531.95,A -85,B 0,C 180,E1 -23891.802,E2 -23891.802} C_VEL
LIN {X 0,Y 182.817,Z 520.846,A -85,B 0,C 180,E1 -23892.47,E2 -23892.47} C_VEL
LIN {X 0,Y 184.402,Z 498.121,A -85,B 0,C 180,E1 -23893.316,E2 -23893.316} C_VEL
LIN {X 0,Y 185.351,Z 481.503,A -85,B 0,C 180,E1 -23893.909,E2 -23893.909} C_VEL
LIN {X 0,Y 184.393,Z 475.364,A -85,B 0,C 180,E1 -23894.52,E2 -23894.52} C_VEL
LIN {X 0,Y 178.982,Z 461.507,A -85,B 0,C 180,E1 -23897.028,E2 -23897.028} C_VEL
LIN {X 0,Y 173.262,Z 449.659,A -85,B 0,C 180,E1 -23899.822,E2 -23899.822} C_VEL
LIN {X 0,Y 169.144,Z 441.869,A -85,B 0,C 180,E1 -23902.013,E2 -23902.013} C_VEL
LIN {X 0,Y 164.831,Z 434.594,A -85,B 0,C 180,E1 -23904.49,E2 -23904.49} C_VEL
LIN {X 0,Y 161.975,Z 430.678,A -85,B 0,C 180,E1 -23906.224,E2 -23906.224} C_VEL
LIN {X 0,Y 159.323,Z 427.309,A -85,B 0,C 180,E1 -23907.944,E2 -23907.944} C_VEL
LIN {X 0,Y 158.466,Z 426.012,A -85,B 0,C 180,E1 -23908.549,E2 -23908.549} C_VEL
LIN {X 0,Y 155.986,Z 423.466,A -85,B 0,C 180,E1 -23910.289,E2 -23910.289} C_VEL
LIN {X 0,Y 154.537,Z 420.94,A -85,B 0,C 180,E1 -23911.475,E2 -23911.475} C_VEL
LIN {X 0,Y 151.905,Z 418.913,A -85,B 0,C 180,E1 -23913.551,E2 -23913.551} C_VEL
LIN {X 0,Y 150.469,Z 416.398,A -85,B 0,C 180,E1 -23915.009,E2 -23915.009} C_VEL
LIN {X 0,Y 150.28,Z 415.502,A -85,B 0,C 180,E1 -23915.844,E2 -23915.844} C_VEL
LIN {X 0,Y 150.365,Z 415.202,A -85,B 0,C 180,E1 -23920.901,E2 -23920.901} C_VEL
LIN {X 0,Y 150.459,Z 415.233,A -85,B 0,C 180,E1 -23926.492,E2 -23926.492} C_VEL
LIN {X 0,Y 150.654,Z 415.165,A -85,B 0,C 180,E1 -23929.244,E2 -23929.244} C_VEL
LIN {X 0,Y 150.741,Z 415.155,A -85,B 0,C 180,E1 -23931.958,E2 -23931.958} C_VEL
LIN {X 0,Y 151.218,Z 415.09,A -85,B 0,C 180,E1 -23939.998,E2 -23939.998} C_VEL
LIN {X 0,Y 150.746,Z 415.163,A -85,B 0,C 180,E1 -23948.038,E2 -23948.038} C_VEL
LIN {X 0,Y 150.609,Z 415.174,A -85,B 0,C 180,E1 -23951.494,E2 -23951.494} C_VEL
LIN {X 0,Y 150.382,Z 415.227,A -85,B 0,C 180,E1 -23956.283,E2 -23956.283} C_VEL
LIN {X 0,Y 150.35,Z 415.214,A -85,B 0,C 180,E1 -23960.79,E2 -23960.79} C_VEL
LIN {X 0,Y 150.263,Z 415.504,A -85,B 0,C 180,E1 -23964.616,E2 -23964.616} C_VEL
LIN {X 0,Y 150.549,Z 416.657,A -85,B 0,C 180,E1 -23965.503,E2 -23965.503} C_VEL
LIN {X 0,Y 152.284,Z 419.374,A -85,B 0,C 180,E1 -23967.165,E2 -23967.165} C_VEL
LIN {X 0,Y 154.803,Z 421.222,A -85,B 0,C 180,E1 -23969.117,E2 -23969.117} C_VEL
LIN {X 0,Y 156.763,Z 424.505,A -85,B 0,C 180,E1 -23970.68,E2 -23970.68} C_VEL
LIN {X 0,Y 158.917,Z 426.559,A -85,B 0,C 180,E1 -23972.147,E2 -23972.147} C_VEL
LIN {X 0,Y 161.511,Z 430.243,A -85,B 0,C 180,E1 -23973.883,E2 -23973.883} C_VEL
LIN {X 0,Y 162.661,Z 431.533,A -85,B 0,C 180,E1 -23974.585,E2 -23974.585} C_VEL
LIN {X 0,Y 166.53,Z 437.007,A -85,B 0,C 180,E1 -23976.873,E2 -23976.873} C_VEL
LIN {X 0,Y 171.871,Z 444.88,A -85,B 0,C 180,E1 -23979.71,E2 -23979.71} C_VEL
LIN {X 0,Y 177.747,Z 454.277,A -85,B 0,C 180,E1 -23982.509,E2 -23982.509} C_VEL
LIN {X 0,Y 183.747,Z 465.452,A -85,B 0,C 180,E1 -23985.134,E2 -23985.134} C_VEL
LIN {X 0,Y 189.629,Z 478.361,A -85,B 0,C 180,E1 -23987.543,E2 -23987.543} C_VEL
LIN {X 0,Y 197.323,Z 495.682,A -85,B 0,C 180,E1 -23990.377,E2 -23990.377} C_VEL
LIN {X 0,Y 205.392,Z 510.051,A -85,B 0,C 180,E1 -23992.909,E2 -23992.909} C_VEL
LIN {X 0,Y 211.817,Z 520.095,A -85,B 0,C 180,E1 -23994.892,E2 -23994.892} C_VEL
LIN {X 0,Y 219.35,Z 530.54,A -85,B 0,C 180,E1 -23997.249,E2 -23997.249} C_VEL
LIN {X 0,Y 227.681,Z 540.729,A -85,B 0,C 180,E1 -23999.8,E2 -23999.8} C_VEL
LIN {X 0,Y 237.428,Z 550.956,A -85,B 0,C 180,E1 -24002.623,E2 -24002.623} C_VEL
LIN {X 0,Y 247.52,Z 559.822,A -85,B 0,C 180,E1 -24005.31,E2 -24005.31} C_VEL
LIN {X 0,Y 257.998,Z 567.577,A -85,B 0,C 180,E1 -24007.844,E2 -24007.844} C_VEL
LIN {X 0,Y 271.469,Z 576.516,A -85,B 0,C 180,E1 -24010.895,E2 -24010.895} C_VEL
LIN {X 0,Y 282.389,Z 583.51,A -85,B 0,C 180,E1 -24013.367,E2 -24013.367} C_VEL
LIN {X 0,Y 287.867,Z 587.035,A -85,B 0,C 180,E1 -24014.65,E2 -24014.65} C_VEL
LIN {X 0,Y 293.537,Z 591.02,A -85,B 0,C 180,E1 -24016.147,E2 -24016.147} C_VEL
LIN {X 0,Y 299.446,Z 594.876,A -85,B 0,C 180,E1 -24017.805,E2 -24017.805} C_VEL
LIN {X 0,Y 304.151,Z 597.841,A -85,B 0,C 180,E1 -24019.347,E2 -24019.347} C_VEL
LIN {X 0,Y 307.595,Z 600.297,A -85,B 0,C 180,E1 -24020.796,E2 -24020.796} C_VEL
LIN {X 0,Y 311.711,Z 602.853,A -85,B 0,C 180,E1 -24022.763,E2 -24022.763} C_VEL
LIN {X 0,Y 315.32,Z 604.776,A -85,B 0,C 180,E1 -24024.885,E2 -24024.885} C_VEL
LIN {X 0,Y 317.083,Z 605.518,A -85,B 0,C 180,E1 -24026.187,E2 -24026.187} C_VEL
LIN {X 0,Y 318.393,Z 606.02,A -85,B 0,C 180,E1 -24027.469,E2 -24027.469} C_VEL
LIN {X 0,Y 319.09,Z 606.346,A -85,B 0,C 180,E1 -24028.738,E2 -24028.738} C_VEL
LIN {X 0,Y 319.445,Z 606.407,A -85,B 0,C 180,E1 -24030,E2 -24030} C_VEL
LIN {X 0,Y 319.107,Z 606.337,A -85,B 0,C 180,E1 -24031.262,E2 -24031.262} C_VEL
LIN {X 0,Y 318.39,Z 606.019,A -85,B 0,C 180,E1 -24032.53,E2 -24032.53} C_VEL
LIN {X 0,Y 316.981,Z 605.501,A -85,B 0,C 180,E1 -24033.878,E2 -24033.878} C_VEL
LIN {X 0,Y 315.296,Z 604.787,A -85,B 0,C 180,E1 -24035.115,E2 -24035.115} C_VEL
LIN {X 0,Y 313.177,Z 603.666,A -85,B 0,C 180,E1 -24036.442,E2 -24036.442} C_VEL
LIN {X 0,Y 310.555,Z 602.24,A -85,B 0,C 180,E1 -24037.803,E2 -24037.803} C_VEL
LIN {X 0,Y 306.549,Z 599.532,A -85,B 0,C 180,E1 -24039.663,E2 -24039.663} C_VEL
LIN {X 0,Y 304.187,Z 597.826,A -85,B 0,C 180,E1 -24040.651,E2 -24040.651} C_VEL
LIN {X 0,Y 298.259,Z 594.17,A -85,B 0,C 180,E1 -24042.541,E2 -24042.541} C_VEL
LIN {X 0,Y 290.565,Z 588.922,A -85,B 0,C 180,E1 -24044.652,E2 -24044.652} C_VEL
LIN {X 0,Y 285.123,Z 585.261,A -85,B 0,C 180,E1 -24045.993,E2 -24045.993} C_VEL
LIN {X 0,Y 274.198,Z 578.232,A -85,B 0,C 180,E1 -24048.498,E2 -24048.498} C_VEL
LIN {X 0,Y 263.35,Z 571.186,A -85,B 0,C 180,E1 -24050.929,E2 -24050.929} C_VEL
LIN {X 0,Y 251.114,Z 562.553,A -85,B 0,C 180,E1 -24053.803,E2 -24053.803} C_VEL
LIN {X 0,Y 240.869,Z 554.132,A -85,B 0,C 180,E1 -24056.447,E2 -24056.447} C_VEL
LIN {X 0,Y 231.662,Z 545.099,A -85,B 0,C 180,E1 -24059.037,E2 -24059.037} C_VEL
LIN {X 0,Y 221.736,Z 533.557,A -85,B 0,C 180,E1 -24062.024,E2 -24062.024} C_VEL
LIN {X 0,Y 213.44,Z 522.496,A -85,B 0,C 180,E1 -24064.597,E2 -24064.597} C_VEL
LIN {X 0,Y 207.095,Z 512.662,A -85,B 0,C 180,E1 -24066.604,E2 -24066.604} C_VEL
LIN {X 0,Y 200.702,Z 501.963,A -85,B 0,C 180,E1 -24068.54,E2 -24068.54} C_VEL
LIN {X 0,Y 194.155,Z 489.028,A -85,B 0,C 180,E1 -24070.725,E2 -24070.725} C_VEL
LIN {X 0,Y 186.364,Z 470.974,A -85,B 0,C 180,E1 -24073.775,E2 -24073.775} C_VEL
LIN {X 0,Y 180.972,Z 460.057,A -85,B 0,C 180,E1 -24076.055,E2 -24076.055} C_VEL
LIN {X 0,Y 175.104,Z 449.921,A -85,B 0,C 180,E1 -24078.715,E2 -24078.715} C_VEL
LIN {X 0,Y 169.698,Z 441.594,A -85,B 0,C 180,E1 -24081.407,E2 -24081.407} C_VEL
LIN {X 0,Y 165.081,Z 434.946,A -85,B 0,C 180,E1 -24083.957,E2 -24083.957} C_VEL
LIN {X 0,Y 161.956,Z 430.676,A -85,B 0,C 180,E1 -24085.848,E2 -24085.848} C_VEL
LIN {X 0,Y 159.222,Z 427.12,A -85,B 0,C 180,E1 -24087.632,E2 -24087.632} C_VEL
LIN {X 0,Y 158.421,Z 425.987,A -85,B 0,C 180,E1 -24088.19,E2 -24088.19} C_VEL
LIN {X 0,Y 155.95,Z 423.429,A -85,B 0,C 180,E1 -24089.929,E2 -24089.929} C_VEL
LIN {X 0,Y 154.517,Z 420.932,A -85,B 0,C 180,E1 -24091.103,E2 -24091.103} C_VEL
LIN {X 0,Y 151.887,Z 418.923,A -85,B 0,C 180,E1 -24093.178,E2 -24093.178} C_VEL
LIN {X 0,Y 150.37,Z 416.012,A -85,B 0,C 180,E1 -24094.862,E2 -24094.862} C_VEL
LIN {X 0,Y 150.262,Z 415.303,A -85,B 0,C 180,E1 -24096.21,E2 -24096.21} C_VEL
LIN {X 0,Y 150.362,Z 415.205,A -85,B 0,C 180,E1 -24100.904,E2 -24100.904} C_VEL
LIN {X 0,Y 150.456,Z 415.221,A -85,B 0,C 180,E1 -24106.495,E2 -24106.495} C_VEL
LIN {X 0,Y 150.647,Z 415.165,A -85,B 0,C 180,E1 -24109.247,E2 -24109.247} C_VEL
LIN {X 0,Y 150.742,Z 415.163,A -85,B 0,C 180,E1 -24111.961,E2 -24111.961} C_VEL
LIN {X 0,Y 151.214,Z 415.091,A -85,B 0,C 180,E1 -24120.002,E2 -24120.002} C_VEL
LIN {X 0,Y 150.737,Z 415.155,A -85,B 0,C 180,E1 -24128.042,E2 -24128.042} C_VEL
LIN {X 0,Y 150.609,Z 415.179,A -85,B 0,C 180,E1 -24131.502,E2 -24131.502} C_VEL
LIN {X 0,Y 150.371,Z 415.214,A -85,B 0,C 180,E1 -24136.287,E2 -24136.287} C_VEL
LIN {X 0,Y 150.349,Z 415.218,A -85,B 0,C 180,E1 -24140.794,E2 -24140.794} C_VEL
LIN {X 0,Y 150.284,Z 415.538,A -85,B 0,C 180,E1 -24144.247,E2 -24144.247} C_VEL
LIN {X 0,Y 150.596,Z 416.748,A -85,B 0,C 180,E1 -24145.167,E2 -24145.167} C_VEL
LIN {X 0,Y 152.155,Z 419.22,A -85,B 0,C 180,E1 -24146.667,E2 -24146.667} C_VEL
LIN {X 0,Y 154.814,Z 421.313,A -85,B 0,C 180,E1 -24148.747,E2 -24148.747} C_VEL
LIN {X 0,Y 156.878,Z 424.62,A -85,B 0,C 180,E1 -24150.375,E2 -24150.375} C_VEL
LIN {X 0,Y 159.044,Z 426.753,A -85,B 0,C 180,E1 -24151.849,E2 -24151.849} C_VEL
LIN {X 0,Y 161.42,Z 430.134,A -85,B 0,C 180,E1 -24153.44,E2 -24153.44} C_VEL
LIN {X 0,Y 162.849,Z 431.793,A -85,B 0,C 180,E1 -24154.315,E2 -24154.315} C_VEL
LIN {X 0,Y 165.915,Z 436.284,A -85,B 0,C 180,E1 -24156.148,E2 -24156.148} C_VEL
LIN {X 0,Y 170.435,Z 444.099,A -85,B 0,C 180,E1 -24158.683,E2 -24158.683} C_VEL
LIN {X 0,Y 177.301,Z 457.858,A -85,B 0,C 180,E1 -24162.175,E2 -24162.175} C_VEL
LIN {X 0,Y 181.916,Z 468.775,A -85,B 0,C 180,E1 -24164.35,E2 -24164.35} C_VEL
LIN {X 0,Y 184.74,Z 476.551,A -85,B 0,C 180,E1 -24165.648,E2 -24165.648} C_VEL
LIN {X 0,Y 185.368,Z 482.518,A -85,B 0,C 180,E1 -24166.15,E2 -24166.15} C_VEL
LIN {X 0,Y 182.926,Z 519.657,A -85,B 0,C 180,E1 -24167.468,E2 -24167.468} C_VEL
LIN {X 0,Y 181.683,Z 530.064,A -85,B 0,C 180,E1 -24168.067,E2 -24168.067} C_VEL
LIN {X 0,Y 180.026,Z 539.444,A -85,B 0,C 180,E1 -24168.795,E2 -24168.795} C_VEL
LIN {X 0,Y 177.971,Z 548.533,A -85,B 0,C 180,E1 -24169.713,E2 -24169.713} C_VEL
LIN {X 0,Y 175.445,Z 557.671,A -85,B 0,C 180,E1 -24170.884,E2 -24170.884} C_VEL
LIN {X 0,Y 172.627,Z 566.669,A -85,B 0,C 180,E1 -24172.363,E2 -24172.363} C_VEL
LIN {X 0,Y 169.509,Z 575.392,A -85,B 0,C 180,E1 -24174.153,E2 -24174.153} C_VEL
LIN {X 0,Y 166.499,Z 582.807,A -85,B 0,C 180,E1 -24175.995,E2 -24175.995} C_VEL
LIN {X 0,Y 162.616,Z 591.599,A -85,B 0,C 180,E1 -24178.762,E2 -24178.762} C_VEL
LIN {X 0,Y 159.844,Z 597.588,A -85,B 0,C 180,E1 -24181.077,E2 -24181.077} C_VEL
LIN {X 0,Y 156.918,Z 603.903,A -85,B 0,C 180,E1 -24184.109,E2 -24184.109} C_VEL
LIN {X 0,Y 154.177,Z 609.174,A -85,B 0,C 180,E1 -24187.204,E2 -24187.204} C_VEL
LIN {X 0,Y 151.549,Z 614.269,A -85,B 0,C 180,E1 -24191.058,E2 -24191.058} C_VEL
LIN {X 0,Y 149.627,Z 618.237,A -85,B 0,C 180,E1 -24195.03,E2 -24195.03} C_VEL
LIN {X 0,Y 148.392,Z 621.179,A -85,B 0,C 180,E1 -24199.081,E2 -24199.081} C_VEL
LIN {X 0,Y 147.901,Z 622.685,A -85,B 0,C 180,E1 -24201.805,E2 -24201.805} C_VEL
LIN {X 0,Y 147.613,Z 624.222,A -85,B 0,C 180,E1 -24207.272,E2 -24207.272} C_VEL
LIN {X 0,Y 147.72,Z 624.506,A -85,B 0,C 180,E1 -24210.001,E2 -24210.001} C_VEL
LIN {X 0,Y 147.625,Z 623.619,A -85,B 0,C 180,E1 -24215.464,E2 -24215.464} C_VEL
LIN {X 0,Y 147.886,Z 622.684,A -85,B 0,C 180,E1 -24218.197,E2 -24218.197} C_VEL
LIN {X 0,Y 149.137,Z 619.327,A -85,B 0,C 180,E1 -24223.629,E2 -24223.629} C_VEL
LIN {X 0,Y 150.812,Z 615.695,A -85,B 0,C 180,E1 -24227.633,E2 -24227.633} C_VEL
LIN {X 0,Y 153.263,Z 610.963,A -85,B 0,C 180,E1 -24231.522,E2 -24231.522} C_VEL
LIN {X 0,Y 156.376,Z 604.993,A -85,B 0,C 180,E1 -24235.275,E2 -24235.275} C_VEL
LIN {X 0,Y 159.113,Z 599.209,A -85,B 0,C 180,E1 -24238.178,E2 -24238.178} C_VEL
LIN {X 0,Y 161.942,Z 593.157,A -85,B 0,C 180,E1 -24240.66,E2 -24240.66} C_VEL
LIN {X 0,Y 164.967,Z 586.504,A -85,B 0,C 180,E1 -24242.901,E2 -24242.901} C_VEL
LIN {X 0,Y 168.204,Z 578.68,A -85,B 0,C 180,E1 -24245.066,E2 -24245.066} C_VEL
LIN {X 0,Y 169.589,Z 575.205,A -85,B 0,C 180,E1 -24245.889,E2 -24245.889} C_VEL
LIN {X 0,Y 170.873,Z 570.553,A -85,B 0,C 180,E1 -24247.033,E2 -24247.033} C_VEL
LIN {X 0,Y 171.29,Z 562.701,A -85,B 0,C 180,E1 -24249.053,E2 -24249.053} C_VEL
LIN {X 0,Y 171.519,Z 554.511,A -85,B 0,C 180,E1 -24250.904,E2 -24250.904} C_VEL
LIN {X 0,Y 172.375,Z 549.155,A -85,B 0,C 180,E1 -24251.72,E2 -24251.72} C_VEL
LIN {X 0,Y 174.735,Z 539.236,A -85,B 0,C 180,E1 -24252.744,E2 -24252.744} C_VEL
LIN {X 0,Y 176.55,Z 529.554,A -85,B 0,C 180,E1 -24253.484,E2 -24253.484} C_VEL
LIN {X 0,Y 177.707,Z 520.223,A -85,B 0,C 180,E1 -24254.029,E2 -24254.029} C_VEL
LIN {X 0,Y 179.694,Z 491.921,A -85,B 0,C 180,E1 -24255.08,E2 -24255.08} C_VEL
LIN {X 0,Y 180.238,Z 482.626,A -85,B 0,C 180,E1 -24255.421,E2 -24255.421} C_VEL
LIN {X 0,Y 179.599,Z 478.482,A -85,B 0,C 180,E1 -24255.859,E2 -24255.859} C_VEL
LIN {X 0,Y 174.681,Z 465.584,A -85,B 0,C 180,E1 -24258.308,E2 -24258.308} C_VEL
LIN {X 0,Y 168.775,Z 452.856,A -85,B 0,C 180,E1 -24261.435,E2 -24261.435} C_VEL
LIN {X 0,Y 164.096,Z 444.188,A -85,B 0,C 180,E1 -24264.144,E2 -24264.144} C_VEL
LIN {X 0,Y 161.551,Z 439.945,A -85,B 0,C 180,E1 -24265.728,E2 -24265.728} C_VEL
LIN {X 0,Y 159.081,Z 436.477,A -85,B 0,C 180,E1 -24267.328,E2 -24267.328} C_VEL
LIN {X 0,Y 156.295,Z 432.567,A -85,B 0,C 180,E1 -24269.285,E2 -24269.285} C_VEL
LIN {X 0,Y 153.286,Z 429.108,A -85,B 0,C 180,E1 -24271.548,E2 -24271.548} C_VEL
LIN {X 0,Y 152.187,Z 427.29,A -85,B 0,C 180,E1 -24272.495,E2 -24272.495} C_VEL
LIN {X 0,Y 149.82,Z 425.236,A -85,B 0,C 180,E1 -24274.494,E2 -24274.494} C_VEL
LIN {X 0,Y 148.136,Z 422.362,A -85,B 0,C 180,E1 -24276.216,E2 -24276.216} C_VEL
LIN {X 0,Y 144.828,Z 419.684,A -85,B 0,C 180,E1 -24279.722,E2 -24279.722} C_VEL
LIN {X 0,Y 143.393,Z 416.717,A -85,B 0,C 180,E1 -24282.16,E2 -24282.16} C_VEL
LIN {X 0,Y 143.341,Z 416.136,A -85,B 0,C 180,E1 -24284.354,E2 -24284.354} C_VEL
LIN {X 0,Y 143.596,Z 416.048,A -85,B 0,C 180,E1 -24288.709,E2 -24288.709} C_VEL
LIN {X 0,Y 143.662,Z 416.033,A -85,B 0,C 180,E1 -24291.559,E2 -24291.559} C_VEL
LIN {X 0,Y 144.177,Z 415.966,A -85,B 0,C 180,E1 -24299.998,E2 -24299.998} C_VEL
LIN {X 0,Y 143.665,Z 416.04,A -85,B 0,C 180,E1 -24308.437,E2 -24308.437} C_VEL
LIN {X 0,Y 143.548,Z 416.054,A -85,B 0,C 180,E1 -24311.711,E2 -24311.711} C_VEL
LIN {X 0,Y 143.328,Z 416.394,A -85,B 0,C 180,E1 -24317.66,E2 -24317.66} C_VEL
LIN {X 0,Y 143.615,Z 417.399,A -85,B 0,C 180,E1 -24318.916,E2 -24318.916} C_VEL
LIN {X 0,Y 145.019,Z 419.913,A -85,B 0,C 180,E1 -24320.897,E2 -24320.897} C_VEL
LIN {X 0,Y 147.477,Z 421.803,A -85,B 0,C 180,E1 -24323.521,E2 -24323.521} C_VEL
LIN {X 0,Y 148.122,Z 422.337,A -85,B 0,C 180,E1 -24324.155,E2 -24324.155} C_VEL
LIN {X 0,Y 150.068,Z 425.566,A -85,B 0,C 180,E1 -24326.124,E2 -24326.124} C_VEL
LIN {X 0,Y 152.622,Z 427.854,A -85,B 0,C 180,E1 -24328.256,E2 -24328.256} C_VEL
LIN {X 0,Y 154.797,Z 431.133,A -85,B 0,C 180,E1 -24330.031,E2 -24330.031} C_VEL
LIN {X 0,Y 156.485,Z 432.892,A -85,B 0,C 180,E1 -24331.245,E2 -24331.245} C_VEL
LIN {X 0,Y 159.28,Z 436.707,A -85,B 0,C 180,E1 -24333.188,E2 -24333.188} C_VEL
LIN {X 0,Y 163.645,Z 442.976,A -85,B 0,C 180,E1 -24335.936,E2 -24335.936} C_VEL
LIN {X 0,Y 168.197,Z 449.793,A -85,B 0,C 180,E1 -24338.5,E2 -24338.5} C_VEL
LIN {X 0,Y 173.959,Z 459.282,A -85,B 0,C 180,E1 -24341.428,E2 -24341.428} C_VEL
LIN {X 0,Y 179.609,Z 470.102,A -85,B 0,C 180,E1 -24344.059,E2 -24344.059} C_VEL
LIN {X 0,Y 185.242,Z 482.851,A -85,B 0,C 180,E1 -24346.517,E2 -24346.517} C_VEL
LIN {X 0,Y 192.595,Z 499.794,A -85,B 0,C 180,E1 -24349.393,E2 -24349.393} C_VEL
LIN {X 0,Y 200.464,Z 514.269,A -85,B 0,C 180,E1 -24352.073,E2 -24352.073} C_VEL
LIN {X 0,Y 208.067,Z 526.515,A -85,B 0,C 180,E1 -24354.73,E2 -24354.73} C_VEL
LIN {X 0,Y 216.382,Z 538.021,A -85,B 0,C 180,E1 -24357.613,E2 -24357.613} C_VEL
LIN {X 0,Y 224.494,Z 547.736,A -85,B 0,C 180,E1 -24360.309,E2 -24360.309} C_VEL
LIN {X 0,Y 232.871,Z 556.349,A -85,B 0,C 180,E1 -24362.911,E2 -24362.911} C_VEL
LIN {X 0,Y 242.878,Z 564.902,A -85,B 0,C 180,E1 -24365.731,E2 -24365.731} C_VEL
LIN {X 0,Y 256.388,Z 574.36,A -85,B 0,C 180,E1 -24369.124,E2 -24369.124} C_VEL
LIN {X 0,Y 269.441,Z 582.471,A -85,B 0,C 180,E1 -24372.18,E2 -24372.18} C_VEL
LIN {X 0,Y 280.411,Z 589.117,A -85,B 0,C 180,E1 -24374.778,E2 -24374.778} C_VEL
LIN {X 0,Y 285.863,Z 592.628,A -85,B 0,C 180,E1 -24376.189,E2 -24376.189} C_VEL
LIN {X 0,Y 291.632,Z 596.401,A -85,B 0,C 180,E1 -24377.79,E2 -24377.79} C_VEL
LIN {X 0,Y 295.731,Z 598.964,A -85,B 0,C 180,E1 -24379.04,E2 -24379.04} C_VEL
LIN {X 0,Y 298.027,Z 600.467,A -85,B 0,C 180,E1 -24379.813,E2 -24379.813} C_VEL
LIN {X 0,Y 302.986,Z 603.892,A -85,B 0,C 180,E1 -24382,E2 -24382} C_VEL
LIN {X 0,Y 305.83,Z 605.567,A -85,B 0,C 180,E1 -24383.402,E2 -24383.402} C_VEL
LIN {X 0,Y 308.153,Z 606.787,A -85,B 0,C 180,E1 -24384.765,E2 -24384.765} C_VEL
LIN {X 0,Y 310.074,Z 607.693,A -85,B 0,C 180,E1 -24386.101,E2 -24386.101} C_VEL
LIN {X 0,Y 311.503,Z 608.251,A -85,B 0,C 180,E1 -24387.413,E2 -24387.413} C_VEL
LIN {X 0,Y 312.31,Z 608.586,A -85,B 0,C 180,E1 -24388.71,E2 -24388.71} C_VEL
LIN {X 0,Y 312.715,Z 608.658,A -85,B 0,C 180,E1 -24390,E2 -24390} C_VEL
LIN {X 0,Y 312.352,Z 608.576,A -85,B 0,C 180,E1 -24391.289,E2 -24391.289} C_VEL
LIN {X 0,Y 311.511,Z 608.253,A -85,B 0,C 180,E1 -24392.586,E2 -24392.586} C_VEL
LIN {X 0,Y 309.969,Z 607.672,A -85,B 0,C 180,E1 -24393.966,E2 -24393.966} C_VEL
LIN {X 0,Y 308.147,Z 606.81,A -85,B 0,C 180,E1 -24395.234,E2 -24395.234} C_VEL
LIN {X 0,Y 304.615,Z 604.878,A -85,B 0,C 180,E1 -24397.221,E2 -24397.221} C_VEL
LIN {X 0,Y 299.807,Z 601.685,A -85,B 0,C 180,E1 -24399.444,E2 -24399.444} C_VEL
LIN {X 0,Y 298.061,Z 600.463,A -85,B 0,C 180,E1 -24400.185,E2 -24400.185} C_VEL
LIN {X 0,Y 291.628,Z 596.432,A -85,B 0,C 180,E1 -24402.199,E2 -24402.199} C_VEL
LIN {X 0,Y 283.138,Z 590.879,A -85,B 0,C 180,E1 -24404.526,E2 -24404.526} C_VEL
LIN {X 0,Y 273.832,Z 585.207,A -85,B 0,C 180,E1 -24406.776,E2 -24406.776} C_VEL
LIN {X 0,Y 263.746,Z 579.071,A -85,B 0,C 180,E1 -24409.129,E2 -24409.129} C_VEL
LIN {X 0,Y 250.6,Z 570.556,A -85,B 0,C 180,E1 -24412.263,E2 -24412.263} C_VEL
LIN {X 0,Y 239.042,Z 561.786,A -85,B 0,C 180,E1 -24415.304,E2 -24415.304} C_VEL
LIN {X 0,Y 229.57,Z 553.154,A -85,B 0,C 180,E1 -24418.083,E2 -24418.083} C_VEL
LIN {X 0,Y 219.816,Z 542.325,A -85,B 0,C 180,E1 -24421.214,E2 -24421.214} C_VEL
LIN {X 0,Y 213.147,Z 533.797,A -85,B 0,C 180,E1 -24423.483,E2 -24423.483} C_VEL
LIN {X 0,Y 205.845,Z 523.186,A -85,B 0,C 180,E1 -24426.029,E2 -24426.029} C_VEL
LIN {X 0,Y 198.745,Z 511.255,A -85,B 0,C 180,E1 -24428.523,E2 -24428.523} C_VEL
LIN {X 0,Y 190.74,Z 495.917,A -85,B 0,C 180,E1 -24431.28,E2 -24431.28} C_VEL
LIN {X 0,Y 181.846,Z 475.005,A -85,B 0,C 180,E1 -24434.943,E2 -24434.943} C_VEL
LIN {X 0,Y 176.576,Z 464.082,A -85,B 0,C 180,E1 -24437.328,E2 -24437.328} C_VEL
LIN {X 0,Y 171.352,Z 454.86,A -85,B 0,C 180,E1 -24439.858,E2 -24439.858} C_VEL
LIN {X 0,Y 165.171,Z 445.005,A -85,B 0,C 180,E1 -24443.19,E2 -24443.19} C_VEL
LIN {X 0,Y 161.294,Z 439.629,A -85,B 0,C 180,E1 -24445.499,E2 -24445.499} C_VEL
LIN {X 0,Y 158.852,Z 436.235,A -85,B 0,C 180,E1 -24447.09,E2 -24447.09} C_VEL
LIN {X 0,Y 155.93,Z 432.179,A -85,B 0,C 180,E1 -24449.158,E2 -24449.158} C_VEL
LIN {X 0,Y 153.315,Z 429.164,A -85,B 0,C 180,E1 -24451.136,E2 -24451.136} C_VEL
LIN {X 0,Y 152.357,Z 427.447,A -85,B 0,C 180,E1 -24451.972,E2 -24451.972} C_VEL
LIN {X 0,Y 149.59,Z 424.97,A -85,B 0,C 180,E1 -24454.321,E2 -24454.321} C_VEL
LIN {X 0,Y 147.808,Z 421.97,A -85,B 0,C 180,E1 -24456.163,E2 -24456.163} C_VEL
LIN {X 0,Y 145.192,Z 420.099,A -85,B 0,C 180,E1 -24458.898,E2 -24458.898} C_VEL
LIN {X 0,Y 143.708,Z 417.667,A -85,B 0,C 180,E1 -24460.912,E2 -24460.912} C_VEL
LIN {X 0,Y 143.351,Z 416.481,A -85,B 0,C 180,E1 -24462.158,E2 -24462.158} C_VEL
LIN {X 0,Y 143.374,Z 416.115,A -85,B 0,C 180,E1 -24465.814,E2 -24465.814} C_VEL
LIN {X 0,Y 143.591,Z 416.046,A -85,B 0,C 180,E1 -24468.711,E2 -24468.711} C_VEL
LIN {X 0,Y 143.661,Z 416.04,A -85,B 0,C 180,E1 -24471.562,E2 -24471.562} C_VEL
LIN {X 0,Y 144.173,Z 415.967,A -85,B 0,C 180,E1 -24480.002,E2 -24480.002} C_VEL
LIN {X 0,Y 143.658,Z 416.034,A -85,B 0,C 180,E1 -24488.441,E2 -24488.441} C_VEL
LIN {X 0,Y 143.546,Z 416.059,A -85,B 0,C 180,E1 -24491.714,E2 -24491.714} C_VEL
LIN {X 0,Y 143.337,Z 416.391,A -85,B 0,C 180,E1 -24497.294,E2 -24497.294} C_VEL
LIN {X 0,Y 143.663,Z 417.608,A -85,B 0,C 180,E1 -24498.635,E2 -24498.635} C_VEL
LIN {X 0,Y 145.312,Z 420.221,A -85,B 0,C 180,E1 -24500.856,E2 -24500.856} C_VEL
LIN {X 0,Y 148.136,Z 422.363,A -85,B 0,C 180,E1 -24503.784,E2 -24503.784} C_VEL
LIN {X 0,Y 149.938,Z 425.408,A -85,B 0,C 180,E1 -24505.618,E2 -24505.618} C_VEL
LIN {X 0,Y 152.547,Z 427.755,A -85,B 0,C 180,E1 -24507.807,E2 -24507.807} C_VEL
LIN {X 0,Y 154.937,Z 431.253,A -85,B 0,C 180,E1 -24509.746,E2 -24509.746} C_VEL
LIN {X 0,Y 156.513,Z 432.962,A -85,B 0,C 180,E1 -24510.882,E2 -24510.882} C_VEL
LIN {X 0,Y 159.27,Z 436.678,A -85,B 0,C 180,E1 -24512.793,E2 -24512.793} C_VEL
LIN {X 0,Y 162.685,Z 441.708,A -85,B 0,C 180,E1 -24514.982,E2 -24514.982} C_VEL
LIN {X 0,Y 166.233,Z 448.019,A -85,B 0,C 180,E1 -24517.125,E2 -24517.125} C_VEL
LIN {X 0,Y 171.429,Z 458.492,A -85,B 0,C 180,E1 -24520.017,E2 -24520.017} C_VEL
LIN {X 0,Y 175.519,Z 467.684,A -85,B 0,C 180,E1 -24522.122,E2 -24522.122} C_VEL
LIN {X 0,Y 179.822,Z 479.204,A -85,B 0,C 180,E1 -24524.254,E2 -24524.254} C_VEL
LIN {X 0,Y 180.206,Z 484.143,A -85,B 0,C 180,E1 -24524.653,E2 -24524.653} C_VEL
LIN {X 0,Y 177.793,Z 519.263,A -85,B 0,C 180,E1 -24525.915,E2 -24525.915} C_VEL
LIN {X 0,Y 176.486,Z 529.568,A -85,B 0,C 180,E1 -24526.498,E2 -24526.498} C_VEL
LIN {X 0,Y 174.763,Z 539.249,A -85,B 0,C 180,E1 -24527.266,E2 -24527.266} C_VEL
LIN {X 0,Y 172.607,Z 548.337,A -85,B 0,C 180,E1 -24528.186,E2 -24528.186} C_VEL
LIN {X 0,Y 170.007,Z 557.477,A -85,B 0,C 180,E1 -24529.377,E2 -24529.377} C_VEL
LIN {X 0,Y 167.055,Z 566.474,A -85,B 0,C 180,E1 -24530.874,E2 -24530.874} C_VEL
LIN {X 0,Y 163.795,Z 575.197,A -85,B 0,C 180,E1 -24532.696,E2 -24532.696} C_VEL
LIN {X 0,Y 160.659,Z 582.612,A -85,B 0,C 180,E1 -24534.578,E2 -24534.578} C_VEL
LIN {X 0,Y 156.576,Z 591.403,A -85,B 0,C 180,E1 -24537.411,E2 -24537.411} C_VEL
LIN {X 0,Y 153.636,Z 597.391,A -85,B 0,C 180,E1 -24539.79,E2 -24539.79} C_VEL
LIN {X 0,Y 150.532,Z 603.707,A -85,B 0,C 180,E1 -24542.923,E2 -24542.923} C_VEL
LIN {X 0,Y 147.626,Z 608.978,A -85,B 0,C 180,E1 -24546.132,E2 -24546.132} C_VEL
LIN {X 0,Y 144.813,Z 614.073,A -85,B 0,C 180,E1 -24550.141,E2 -24550.141} C_VEL
LIN {X 0,Y 142.729,Z 618.041,A -85,B 0,C 180,E1 -24554.288,E2 -24554.288} C_VEL
LIN {X 0,Y 141.402,Z 620.984,A -85,B 0,C 180,E1 -24558.534,E2 -24558.534} C_VEL
LIN {X 0,Y 140.852,Z 622.49,A -85,B 0,C 180,E1 -24561.392,E2 -24561.392} C_VEL
LIN {X 0,Y 140.617,Z 623.426,A -85,B 0,C 180,E1 -24564.264,E2 -24564.264} C_VEL
LIN {X 0,Y 140.632,Z 624.311,A -85,B 0,C 180,E1 -24570.001,E2 -24570.001} C_VEL
LIN {X 0,Y 140.549,Z 623.423,A -85,B 0,C 180,E1 -24575.74,E2 -24575.74} C_VEL
LIN {X 0,Y 140.841,Z 622.489,A -85,B 0,C 180,E1 -24578.61,E2 -24578.61} C_VEL
LIN {X 0,Y 142.221,Z 619.131,A -85,B 0,C 180,E1 -24584.306,E2 -24584.306} C_VEL
LIN {X 0,Y 144.023,Z 615.499,A -85,B 0,C 180,E1 -24588.493,E2 -24588.493} C_VEL
LIN {X 0,Y 146.633,Z 610.767,A -85,B 0,C 180,E1 -24592.547,E2 -24592.547} C_VEL
LIN {X 0,Y 149.946,Z 604.797,A -85,B 0,C 180,E1 -24596.441,E2 -24596.441} C_VEL
LIN {X 0,Y 152.726,Z 599.28,A -85,B 0,C 180,E1 -24599.316,E2 -24599.316} C_VEL
LIN {X 0,Y 155.848,Z 592.961,A -85,B 0,C 180,E1 -24601.997,E2 -24601.997} C_VEL
LIN {X 0,Y 159.051,Z 586.309,A -85,B 0,C 180,E1 -24604.291,E2 -24604.291} C_VEL
LIN {X 0,Y 162.429,Z 578.484,A -85,B 0,C 180,E1 -24606.508,E2 -24606.508} C_VEL
LIN {X 0,Y 165.674,Z 570.406,A -85,B 0,C 180,E1 -24608.346,E2 -24608.346} C_VEL
LIN {X 0,Y 169.044,Z 560.649,A -85,B 0,C 180,E1 -24610.122,E2 -24610.122} C_VEL
LIN {X 0,Y 171.539,Z 552.261,A -85,B 0,C 180,E1 -24611.349,E2 -24611.349} C_VEL
LIN {X 0,Y 172.375,Z 549.155,A -85,B 0,C 180,E1 -24611.72,E2 -24611.72} C_VEL
LIN {X 0,Y 173.233,Z 543.827,A -85,B 0,C 180,E1 -24612.481,E2 -24612.481} C_VEL
LIN {X 0,Y 173.028,Z 534.861,A -85,B 0,C 180,E1 -24613.944,E2 -24613.944} C_VEL
LIN {X 0,Y 172.52,Z 525.733,A -85,B 0,C 180,E1 -24615.216,E2 -24615.216} C_VEL
LIN {X 0,Y 172.689,Z 519.982,A -85,B 0,C 180,E1 -24615.665,E2 -24615.665} C_VEL
LIN {X 0,Y 174.886,Z 490.09,A -85,B 0,C 180,E1 -24616.779,E2 -24616.779} C_VEL
LIN {X 0,Y 175.25,Z 483.847,A -85,B 0,C 180,E1 -24617.018,E2 -24617.018} C_VEL
LIN {X 0,Y 174.513,Z 480.408,A -85,B 0,C 180,E1 -24617.481,E2 -24617.481} C_VEL
LIN {X 0,Y 169.482,Z 467.265,A -85,B 0,C 180,E1 -24620.198,E2 -24620.198} C_VEL
LIN {X 0,Y 163.296,Z 454.022,A -85,B 0,C 180,E1 -24623.811,E2 -24623.811} C_VEL
LIN {X 0,Y 159.048,Z 446.16,A -85,B 0,C 180,E1 -24626.565,E2 -24626.565} C_VEL
LIN {X 0,Y 156.16,Z 442.144,A -85,B 0,C 180,E1 -24628.537,E2 -24628.537} C_VEL
LIN {X 0,Y 153.299,Z 438.191,A -85,B 0,C 180,E1 -24630.682,E2 -24630.682} C_VEL
LIN {X 0,Y 150.429,Z 434.31,A -85,B 0,C 180,E1 -24633.07,E2 -24633.07} C_VEL
LIN {X 0,Y 146.927,Z 430.347,A -85,B 0,C 180,E1 -24636.336,E2 -24636.336} C_VEL
LIN {X 0,Y 146.033,Z 428.63,A -85,B 0,C 180,E1 -24637.354,E2 -24637.354} C_VEL
LIN {X 0,Y 143.395,Z 426.507,A -85,B 0,C 180,E1 -24640.307,E2 -24640.307} C_VEL
LIN {X 0,Y 141.542,Z 423.247,A -85,B 0,C 180,E1 -24643.038,E2 -24643.038} C_VEL
LIN {X 0,Y 138.4,Z 420.924,A -85,B 0,C 180,E1 -24648.503,E2 -24648.503} C_VEL
LIN {X 0,Y 136.737,Z 417.673,A -85,B 0,C 180,E1 -24654.838,E2 -24654.838} C_VEL
LIN {X 0,Y 137.134,Z 416.975,A -85,B 0,C 180,E1 -24659.998,E2 -24659.998} C_VEL
LIN {X 0,Y 136.721,Z 417.592,A -85,B 0,C 180,E1 -24665.159,E2 -24665.159} C_VEL
LIN {X 0,Y 137.458,Z 419.574,A -85,B 0,C 180,E1 -24669.378,E2 -24669.378} C_VEL
LIN {X 0,Y 139.947,Z 422.351,A -85,B 0,C 180,E1 -24674.912,E2 -24674.912} C_VEL
LIN {X 0,Y 141.648,Z 423.344,A -85,B 0,C 180,E1 -24677.504,E2 -24677.504} C_VEL
LIN {X 0,Y 143.385,Z 426.479,A -85,B 0,C 180,E1 -24680.064,E2 -24680.064} C_VEL
LIN {X 0,Y 145.697,Z 428.475,A -85,B 0,C 180,E1 -24682.698,E2 -24682.698} C_VEL
LIN {X 0,Y 146.373,Z 429.294,A -85,B 0,C 180,E1 -24683.428,E2 -24683.428} C_VEL
LIN {X 0,Y 148.614,Z 432.557,A -85,B 0,C 180,E1 -24685.725,E2 -24685.725} C_VEL
LIN {X 0,Y 150.394,Z 434.234,A -85,B 0,C 180,E1 -24687.282,E2 -24687.282} C_VEL
LIN {X 0,Y 152.968,Z 437.86,A -85,B 0,C 180,E1 -24689.454,E2 -24689.454} C_VEL
LIN {X 0,Y 154.105,Z 439.232,A -85,B 0,C 180,E1 -24690.324,E2 -24690.324} C_VEL
LIN {X 0,Y 157.77,Z 444.422,A -85,B 0,C 180,E1 -24692.975,E2 -24692.975} C_VEL
LIN {X 0,Y 162.141,Z 450.801,A -85,B 0,C 180,E1 -24695.779,E2 -24695.779} C_VEL
LIN {X 0,Y 168.395,Z 461.01,A -85,B 0,C 180,E1 -24699.333,E2 -24699.333} C_VEL
LIN {X 0,Y 174.424,Z 472.416,A -85,B 0,C 180,E1 -24702.396,E2 -24702.396} C_VEL
LIN {X 0,Y 179.899,Z 484.81,A -85,B 0,C 180,E1 -24704.978,E2 -24704.978} C_VEL
LIN {X 0,Y 187.846,Z 503.71,A -85,B 0,C 180,E1 -24708.328,E2 -24708.328} C_VEL
LIN {X 0,Y 195.335,Z 518.178,A -85,B 0,C 180,E1 -24711.183,E2 -24711.183} C_VEL
LIN {X 0,Y 201.494,Z 528.788,A -85,B 0,C 180,E1 -24713.633,E2 -24713.633} C_VEL
LIN {X 0,Y 208.656,Z 539.404,A -85,B 0,C 180,E1 -24716.427,E2 -24716.427} C_VEL
LIN {X 0,Y 216.499,Z 549.41,A -85,B 0,C 180,E1 -24719.341,E2 -24719.341} C_VEL
LIN {X 0,Y 225.766,Z 559.324,A -85,B 0,C 180,E1 -24722.518,E2 -24722.518} C_VEL
LIN {X 0,Y 235.539,Z 567.826,A -85,B 0,C 180,E1 -24725.508,E2 -24725.508} C_VEL
LIN {X 0,Y 248.467,Z 576.863,A -85,B 0,C 180,E1 -24728.972,E2 -24728.972} C_VEL
LIN {X 0,Y 262.869,Z 585.503,A -85,B 0,C 180,E1 -24732.496,E2 -24732.496} C_VEL
LIN {X 0,Y 273.68,Z 591.633,A -85,B 0,C 180,E1 -24735.12,E2 -24735.12} C_VEL
LIN {X 0,Y 281.172,Z 596.117,A -85,B 0,C 180,E1 -24737.111,E2 -24737.111} C_VEL
LIN {X 0,Y 289.334,Z 601.021,A -85,B 0,C 180,E1 -24739.503,E2 -24739.503} C_VEL
LIN {X 0,Y 292.155,Z 602.814,A -85,B 0,C 180,E1 -24740.494,E2 -24740.494} C_VEL
LIN {X 0,Y 295.172,Z 604.917,A -85,B 0,C 180,E1 -24741.786,E2 -24741.786} C_VEL
LIN {X 0,Y 298.266,Z 606.86,A -85,B 0,C 180,E1 -24743.234,E2 -24743.234} C_VEL
LIN {X 0,Y 300.744,Z 608.217,A -85,B 0,C 180,E1 -24744.636,E2 -24744.636} C_VEL
LIN {X 0,Y 302.913,Z 609.276,A -85,B 0,C 180,E1 -24746.066,E2 -24746.066} C_VEL
LIN {X 0,Y 304.447,Z 609.944,A -85,B 0,C 180,E1 -24747.353,E2 -24747.353} C_VEL
LIN {X 0,Y 305.387,Z 610.339,A -85,B 0,C 180,E1 -24748.681,E2 -24748.681} C_VEL
LIN {X 0,Y 305.853,Z 610.427,A -85,B 0,C 180,E1 -24750,E2 -24750} C_VEL
LIN {X 0,Y 305.419,Z 610.335,A -85,B 0,C 180,E1 -24751.318,E2 -24751.318} C_VEL
LIN {X 0,Y 304.448,Z 609.953,A -85,B 0,C 180,E1 -24752.646,E2 -24752.646} C_VEL
LIN {X 0,Y 302.814,Z 609.263,A -85,B 0,C 180,E1 -24753.992,E2 -24753.992} C_VEL
LIN {X 0,Y 300.745,Z 608.249,A -85,B 0,C 180,E1 -24755.363,E2 -24755.363} C_VEL
LIN {X 0,Y 297.466,Z 606.43,A -85,B 0,C 180,E1 -24757.122,E2 -24757.122} C_VEL
LIN {X 0,Y 293.696,Z 603.896,A -85,B 0,C 180,E1 -24758.861,E2 -24758.861} C_VEL
LIN {X 0,Y 291.689,Z 602.447,A -85,B 0,C 180,E1 -24759.709,E2 -24759.709} C_VEL
LIN {X 0,Y 286.651,Z 599.409,A -85,B 0,C 180,E1 -24761.311,E2 -24761.311} C_VEL
LIN {X 0,Y 278.187,Z 594.305,A -85,B 0,C 180,E1 -24763.703,E2 -24763.703} C_VEL
LIN {X 0,Y 270.15,Z 589.681,A -85,B 0,C 180,E1 -24765.731,E2 -24765.731} C_VEL
LIN {X 0,Y 261.032,Z 584.469,A -85,B 0,C 180,E1 -24767.944,E2 -24767.944} C_VEL
LIN {X 0,Y 248.45,Z 576.912,A -85,B 0,C 180,E1 -24771.018,E2 -24771.018} C_VEL
LIN {X 0,Y 235.548,Z 567.799,A -85,B 0,C 180,E1 -24774.497,E2 -24774.497} C_VEL
LIN {X 0,Y 225.768,Z 559.319,A -85,B 0,C 180,E1 -24777.483,E2 -24777.483} C_VEL
LIN {X 0,Y 217.643,Z 550.685,A -85,B 0,C 180,E1 -24780.257,E2 -24780.257} C_VEL
LIN {X 0,Y 209.801,Z 540.976,A -85,B 0,C 180,E1 -24783.129,E2 -24783.129} C_VEL
LIN {X 0,Y 203.243,Z 531.625,A -85,B 0,C 180,E1 -24785.652,E2 -24785.652} C_VEL
LIN {X 0,Y 197.75,Z 522.425,A -85,B 0,C 180,E1 -24787.849,E2 -24787.849} C_VEL
LIN {X 0,Y 192.332,Z 512.551,A -85,B 0,C 180,E1 -24789.987,E2 -24789.987} C_VEL
LIN {X 0,Y 185.517,Z 498.69,A -85,B 0,C 180,E1 -24792.579,E2 -24792.579} C_VEL
LIN {X 0,Y 177.409,Z 478.979,A -85,B 0,C 180,E1 -24796.172,E2 -24796.172} C_VEL
LIN {X 0,Y 172.556,Z 468.69,A -85,B 0,C 180,E1 -24798.522,E2 -24798.522} C_VEL
LIN {X 0,Y 167.328,Z 459.269,A -85,B 0,C 180,E1 -24801.235,E2 -24801.235} C_VEL
LIN {X 0,Y 161.901,Z 450.401,A -85,B 0,C 180,E1 -24804.37,E2 -24804.37} C_VEL
LIN {X 0,Y 156.606,Z 442.649,A -85,B 0,C 180,E1 -24807.844,E2 -24807.844} C_VEL
LIN {X 0,Y 153.309,Z 438.203,A -85,B 0,C 180,E1 -24810.288,E2 -24810.288} C_VEL
LIN {X 0,Y 150.736,Z 434.849,A -85,B 0,C 180,E1 -24812.402,E2 -24812.402} C_VEL
LIN {X 0,Y 149.989,Z 433.714,A -85,B 0,C 180,E1 -24813.075,E2 -24813.075} C_VEL
LIN {X 0,Y 147.375,Z 431.021,A -85,B 0,C 180,E1 -24815.48,E2 -24815.48} C_VEL
LIN {X 0,Y 146.016,Z 428.647,A -85,B 0,C 180,E1 -24816.981,E2 -24816.981} C_VEL
LIN {X 0,Y 143.382,Z 426.507,A -85,B 0,C 180,E1 -24819.935,E2 -24819.935} C_VEL
LIN {X 0,Y 141.531,Z 423.232,A -85,B 0,C 180,E1 -24822.668,E2 -24822.668} C_VEL
LIN {X 0,Y 138.327,Z 420.88,A -85,B 0,C 180,E1 -24828.276,E2 -24828.276} C_VEL
LIN {X 0,Y 136.732,Z 417.82,A -85,B 0,C 180,E1 -24834.101,E2 -24834.101} C_VEL
LIN {X 0,Y 136.794,Z 417.202,A -85,B 0,C 180,E1 -24837.057,E2 -24837.057} C_VEL
LIN {X 0,Y 137.13,Z 416.974,A -85,B 0,C 180,E1 -24840.002,E2 -24840.002} C_VEL
LIN {X 0,Y 136.733,Z 417.695,A -85,B 0,C 180,E1 -24845.162,E2 -24845.162} C_VEL
LIN {X 0,Y 138,Z 420.422,A -85,B 0,C 180,E1 -24850.528,E2 -24850.528} C_VEL
LIN {X 0,Y 140.388,Z 422.58,A -85,B 0,C 180,E1 -24855.239,E2 -24855.239} C_VEL
LIN {X 0,Y 141.711,Z 423.471,A -85,B 0,C 180,E1 -24857.22,E2 -24857.22} C_VEL
LIN {X 0,Y 143.394,Z 426.512,A -85,B 0,C 180,E1 -24859.693,E2 -24859.693} C_VEL
LIN {X 0,Y 146.244,Z 429.035,A -85,B 0,C 180,E1 -24862.891,E2 -24862.891} C_VEL
LIN {X 0,Y 148.482,Z 432.403,A -85,B 0,C 180,E1 -24865.215,E2 -24865.215} C_VEL
LIN {X 0,Y 150.49,Z 434.413,A -85,B 0,C 180,E1 -24866.986,E2 -24866.986} C_VEL
LIN {X 0,Y 153.245,Z 438.131,A -85,B 0,C 180,E1 -24869.277,E2 -24869.277} C_VEL
LIN {X 0,Y 157.629,Z 444.135,A -85,B 0,C 180,E1 -24872.484,E2 -24872.484} C_VEL
LIN {X 0,Y 159.963,Z 447.898,A -85,B 0,C 180,E1 -24874.061,E2 -24874.061} C_VEL
LIN {X 0,Y 163.73,Z 454.92,A -85,B 0,C 180,E1 -24876.46,E2 -24876.46} C_VEL
LIN {X 0,Y 169.64,Z 467.66,A -85,B 0,C 180,E1 -24879.891,E2 -24879.891} C_VEL
LIN {X 0,Y 174.508,Z 480.454,A -85,B 0,C 180,E1 -24882.52,E2 -24882.52} C_VEL
LIN {X 0,Y 175.077,Z 482.436,A -85,B 0,C 180,E1 -24882.838,E2 -24882.838} C_VEL
LIN {X 0,Y 175.182,Z 485.689,A -85,B 0,C 180,E1 -24883.066,E2 -24883.066} C_VEL
LIN {X 0,Y 172.669,Z 519.982,A -85,B 0,C 180,E1 -24884.32,E2 -24884.32} C_VEL
LIN {X 0,Y 171.053,Z 531.65,A -85,B 0,C 180,E1 -24885.021,E2 -24885.021} C_VEL
LIN {X 0,Y 168.206,Z 545.183,A -85,B 0,C 180,E1 -24886.212,E2 -24886.212} C_VEL
LIN {X 0,Y 164.698,Z 557.282,A -85,B 0,C 180,E1 -24887.773,E2 -24887.773} C_VEL
LIN {X 0,Y 161.611,Z 566.279,A -85,B 0,C 180,E1 -24889.286,E2 -24889.286} C_VEL
LIN {X 0,Y 158.194,Z 575.001,A -85,B 0,C 180,E1 -24891.134,E2 -24891.134} C_VEL
LIN {X 0,Y 154.93,Z 582.417,A -85,B 0,C 180,E1 -24893.056,E2 -24893.056} C_VEL
LIN {X 0,Y 150.62,Z 591.208,A -85,B 0,C 180,E1 -24895.951,E2 -24895.951} C_VEL
LIN {X 0,Y 147.517,Z 597.196,A -85,B 0,C 180,E1 -24898.396,E2 -24898.396} C_VEL
LIN {X 0,Y 144.478,Z 603.022,A -85,B 0,C 180,E1 -24901.335,E2 -24901.335} C_VEL
LIN {X 0,Y 141.141,Z 608.783,A -85,B 0,C 180,E1 -24904.961,E2 -24904.961} C_VEL
LIN {X 0,Y 138.127,Z 613.877,A -85,B 0,C 180,E1 -24909.136,E2 -24909.136} C_VEL
LIN {X 0,Y 135.87,Z 617.845,A -85,B 0,C 180,E1 -24913.473,E2 -24913.473} C_VEL
LIN {X 0,Y 134.437,Z 620.788,A -85,B 0,C 180,E1 -24917.931,E2 -24917.931} C_VEL
LIN {X 0,Y 133.826,Z 622.294,A -85,B 0,C 180,E1 -24920.936,E2 -24920.936} C_VEL
LIN {X 0,Y 133.414,Z 623.831,A -85,B 0,C 180,E1 -24926.981,E2 -24926.981} C_VEL
LIN {X 0,Y 133.536,Z 624.116,A -85,B 0,C 180,E1 -24930.001,E2 -24930.001} C_VEL
LIN {X 0,Y 133.466,Z 623.228,A -85,B 0,C 180,E1 -24936.046,E2 -24936.046} C_VEL
LIN {X 0,Y 133.817,Z 622.293,A -85,B 0,C 180,E1 -24939.066,E2 -24939.066} C_VEL
LIN {X 0,Y 135.328,Z 618.936,A -85,B 0,C 180,E1 -24945.051,E2 -24945.051} C_VEL
LIN {X 0,Y 137.276,Z 615.303,A -85,B 0,C 180,E1 -24949.438,E2 -24949.438} C_VEL
LIN {X 0,Y 140.058,Z 610.57,A -85,B 0,C 180,E1 -24953.669,E2 -24953.669} C_VEL
LIN {X 0,Y 143.592,Z 604.601,A -85,B 0,C 180,E1 -24957.709,E2 -24957.709} C_VEL
LIN {X 0,Y 146.869,Z 598.508,A -85,B 0,C 180,E1 -24960.958,E2 -24960.958} C_VEL
LIN {X 0,Y 149.861,Z 592.765,A -85,B 0,C 180,E1 -24963.439,E2 -24963.439} C_VEL
LIN {X 0,Y 153.227,Z 586.113,A -85,B 0,C 180,E1 -24965.789,E2 -24965.789} C_VEL
LIN {X 0,Y 156.761,Z 578.288,A -85,B 0,C 180,E1 -24968.058,E2 -24968.058} C_VEL
LIN {X 0,Y 160.148,Z 570.21,A -85,B 0,C 180,E1 -24969.927,E2 -24969.927} C_VEL
LIN {X 0,Y 163.667,Z 560.453,A -85,B 0,C 180,E1 -24971.727,E2 -24971.727} C_VEL
LIN {X 0,Y 166.282,Z 552.067,A -85,B 0,C 180,E1 -24972.964,E2 -24972.964} C_VEL
LIN {X 0,Y 169.049,Z 541.566,A -85,B 0,C 180,E1 -24974.136,E2 -24974.136} C_VEL
LIN {X 0,Y 171.106,Z 531.637,A -85,B 0,C 180,E1 -24974.963,E2 -24974.963} C_VEL
LIN {X 0,Y 172.61,Z 520.789,A -85,B 0,C 180,E1 -24975.628,E2 -24975.628} C_VEL
LIN {X 0,Y 172.689,Z 519.982,A -85,B 0,C 180,E1 -24975.665,E2 -24975.665} C_VEL
LIN {X 0,Y 172.811,Z 514.207,A -85,B 0,C 180,E1 -24976.077,E2 -24976.077} C_VEL
LIN {X 0,Y 170.184,Z 495.553,A -85,B 0,C 180,E1 -24978.148,E2 -24978.148} C_VEL
LIN {X 0,Y 170.1,Z 489.75,A -85,B 0,C 180,E1 -24978.532,E2 -24978.532} C_VEL
LIN {X 0,Y 170.402,Z 485.108,A -85,B 0,C 180,E1 -24978.706,E2 -24978.706} C_VEL
LIN {X 0,Y 166.386,Z 473.71,A -85,B 0,C 180,E1 -24981.052,E2 -24981.052} C_VEL
LIN {X 0,Y 160.581,Z 460.563,A -85,B 0,C 180,E1 -24984.651,E2 -24984.651} C_VEL
LIN {X 0,Y 156.968,Z 453.474,A -85,B 0,C 180,E1 -24987.119,E2 -24987.119} C_VEL
LIN {X 0,Y 154.289,Z 448.95,A -85,B 0,C 180,E1 -24989.076,E2 -24989.076} C_VEL
LIN {X 0,Y 150.735,Z 444.122,A -85,B 0,C 180,E1 -24991.863,E2 -24991.863} C_VEL
LIN {X 0,Y 147.82,Z 440.058,A -85,B 0,C 180,E1 -24994.478,E2 -24994.478} C_VEL
LIN {X 0,Y 145.097,Z 436.89,A -85,B 0,C 180,E1 -24997.2,E2 -24997.2} C_VEL
LIN {X 0,Y 143.999,Z 435.172,A -85,B 0,C 180,E1 -24998.478,E2 -24998.478} C_VEL
LIN {X 0,Y 141.277,Z 432.37,A -85,B 0,C 180,E1 -25001.884,E2 -25001.884} C_VEL
LIN {X 0,Y 140.002,Z 429.901,A -85,B 0,C 180,E1 -25003.971,E2 -25003.971} C_VEL
LIN {X 0,Y 137.439,Z 428.026,A -85,B 0,C 180,E1 -25008.648,E2 -25008.648} C_VEL
LIN {X 0,Y 135.533,Z 424.541,A -85,B 0,C 180,E1 -25015.537,E2 -25015.537} C_VEL
LIN {X 0,Y 135.176,Z 423.81,A -85,B 0,C 180,E1 -25019.998,E2 -25019.998} C_VEL
LIN {X 0,Y 135.65,Z 424.808,A -85,B 0,C 180,E1 -25025.573,E2 -25025.573} C_VEL
LIN {X 0,Y 138.597,Z 429.135,A -85,B 0,C 180,E1 -25034.123,E2 -25034.123} C_VEL
LIN {X 0,Y 140.234,Z 430.216,A -85,B 0,C 180,E1 -25036.794,E2 -25036.794} C_VEL
LIN {X 0,Y 141.999,Z 433.372,A -85,B 0,C 180,E1 -25039.515,E2 -25039.515} C_VEL
LIN {X 0,Y 144.533,Z 435.824,A -85,B 0,C 180,E1 -25042.517,E2 -25042.517} C_VEL
LIN {X 0,Y 146.956,Z 439.293,A -85,B 0,C 180,E1 -25045.113,E2 -25045.113} C_VEL
LIN {X 0,Y 148.269,Z 440.645,A -85,B 0,C 180,E1 -25046.33,E2 -25046.33} C_VEL
LIN {X 0,Y 150.944,Z 444.359,A -85,B 0,C 180,E1 -25048.694,E2 -25048.694} C_VEL
LIN {X 0,Y 155.266,Z 450.605,A -85,B 0,C 180,E1 -25052.045,E2 -25052.045} C_VEL
LIN {X 0,Y 159.314,Z 456.778,A -85,B 0,C 180,E1 -25054.799,E2 -25054.799} C_VEL
LIN {X 0,Y 164.899,Z 466.215,A -85,B 0,C 180,E1 -25058.178,E2 -25058.178} C_VEL
LIN {X 0,Y 170.43,Z 477.003,A -85,B 0,C 180,E1 -25061.184,E2 -25061.184} C_VEL
LIN {X 0,Y 175.565,Z 489.016,A -85,B 0,C 180,E1 -25063.779,E2 -25063.779} C_VEL
LIN {X 0,Y 183.019,Z 507.317,A -85,B 0,C 180,E1 -25067.154,E2 -25067.154} C_VEL
LIN {X 0,Y 188.885,Z 519.535,A -85,B 0,C 180,E1 -25069.706,E2 -25069.706} C_VEL
LIN {X 0,Y 193.942,Z 529.035,A -85,B 0,C 180,E1 -25071.972,E2 -25071.972} C_VEL
LIN {X 0,Y 200.146,Z 539.235,A -85,B 0,C 180,E1 -25074.725,E2 -25074.725} C_VEL
LIN {X 0,Y 206.172,Z 547.788,A -85,B 0,C 180,E1 -25077.268,E2 -25077.268} C_VEL
LIN {X 0,Y 214.505,Z 557.837,A -85,B 0,C 180,E1 -25080.563,E2 -25080.563} C_VEL
LIN {X 0,Y 224.152,Z 567.24,A -85,B 0,C 180,E1 -25083.963,E2 -25083.963} C_VEL
LIN {X 0,Y 234.067,Z 575.003,A -85,B 0,C 180,E1 -25087.025,E2 -25087.025} C_VEL
LIN {X 0,Y 246.282,Z 582.773,A -85,B 0,C 180,E1 -25090.336,E2 -25090.336} C_VEL
LIN {X 0,Y 259.146,Z 589.907,A -85,B 0,C 180,E1 -25093.555,E2 -25093.555} C_VEL
LIN {X 0,Y 268.206,Z 594.697,A -85,B 0,C 180,E1 -25095.818,E2 -25095.818} C_VEL
LIN {X 0,Y 273.747,Z 597.735,A -85,B 0,C 180,E1 -25097.309,E2 -25097.309} C_VEL
LIN {X 0,Y 279.296,Z 600.832,A -85,B 0,C 180,E1 -25098.917,E2 -25098.917} C_VEL
LIN {X 0,Y 284.881,Z 603.915,A -85,B 0,C 180,E1 -25100.674,E2 -25100.674} C_VEL
LIN {X 0,Y 288.785,Z 606.456,A -85,B 0,C 180,E1 -25102.308,E2 -25102.308} C_VEL
LIN {X 0,Y 293.129,Z 609.08,A -85,B 0,C 180,E1 -25104.496,E2 -25104.496} C_VEL
LIN {X 0,Y 295.829,Z 610.474,A -85,B 0,C 180,E1 -25106.179,E2 -25106.179} C_VEL
LIN {X 0,Y 297.203,Z 611.098,A -85,B 0,C 180,E1 -25107.289,E2 -25107.289} C_VEL
LIN {X 0,Y 298.311,Z 611.516,A -85,B 0,C 180,E1 -25108.65,E2 -25108.65} C_VEL
LIN {X 0,Y 298.862,Z 611.62,A -85,B 0,C 180,E1 -25110,E2 -25110} C_VEL
LIN {X 0,Y 298.336,Z 611.52,A -85,B 0,C 180,E1 -25111.349,E2 -25111.349} C_VEL
LIN {X 0,Y 297.205,Z 611.114,A -85,B 0,C 180,E1 -25112.71,E2 -25112.71} C_VEL
LIN {X 0,Y 295.401,Z 610.311,A -85,B 0,C 180,E1 -25114.092,E2 -25114.092} C_VEL
LIN {X 0,Y 293.12,Z 609.089,A -85,B 0,C 180,E1 -25115.503,E2 -25115.503} C_VEL
LIN {X 0,Y 290.288,Z 607.471,A -85,B 0,C 180,E1 -25116.97,E2 -25116.97} C_VEL
LIN {X 0,Y 287.066,Z 605.343,A -85,B 0,C 180,E1 -25118.446,E2 -25118.446} C_VEL
LIN {X 0,Y 284.884,Z 603.908,A -85,B 0,C 180,E1 -25119.33,E2 -25119.33} C_VEL
LIN {X 0,Y 279.295,Z 600.835,A -85,B 0,C 180,E1 -25121.081,E2 -25121.081} C_VEL
LIN {X 0,Y 270.751,Z 596.094,A -85,B 0,C 180,E1 -25123.509,E2 -25123.509} C_VEL
LIN {X 0,Y 261.118,Z 591.024,A -85,B 0,C 180,E1 -25125.946,E2 -25125.946} C_VEL
LIN {X 0,Y 248.969,Z 584.338,A -85,B 0,C 180,E1 -25128.98,E2 -25128.98} C_VEL
LIN {X 0,Y 235.784,Z 576.2,A -85,B 0,C 180,E1 -25132.482,E2 -25132.482} C_VEL
LIN {X 0,Y 224.15,Z 567.245,A -85,B 0,C 180,E1 -25136.036,E2 -25136.036} C_VEL
LIN {X 0,Y 215.155,Z 558.508,A -85,B 0,C 180,E1 -25139.196,E2 -25139.196} C_VEL
LIN {X 0,Y 207.538,Z 549.562,A -85,B 0,C 180,E1 -25142.159,E2 -25142.159} C_VEL
LIN {X 0,Y 200.13,Z 539.298,A -85,B 0,C 180,E1 -25145.269,E2 -25145.269} C_VEL
LIN {X 0,Y 193.937,Z 529.047,A -85,B 0,C 180,E1 -25148.027,E2 -25148.027} C_VEL
LIN {X 0,Y 187.5,Z 516.719,A -85,B 0,C 180,E1 -25150.932,E2 -25150.932} C_VEL
LIN {X 0,Y 181.557,Z 504.112,A -85,B 0,C 180,E1 -25153.455,E2 -25153.455} C_VEL
LIN {X 0,Y 173.191,Z 483.314,A -85,B 0,C 180,E1 -25157.395,E2 -25157.395} C_VEL
LIN {X 0,Y 168.634,Z 473.308,A -85,B 0,C 180,E1 -25159.763,E2 -25159.763} C_VEL
LIN {X 0,Y 163.852,Z 464.416,A -85,B 0,C 180,E1 -25162.42,E2 -25162.42} C_VEL
LIN {X 0,Y 158.888,Z 456.066,A -85,B 0,C 180,E1 -25165.48,E2 -25165.48} C_VEL
LIN {X 0,Y 153.777,Z 448.359,A -85,B 0,C 180,E1 -25169.06,E2 -25169.06} C_VEL
LIN {X 0,Y 150.755,Z 444.173,A -85,B 0,C 180,E1 -25171.457,E2 -25171.457} C_VEL
LIN {X 0,Y 147.664,Z 439.928,A -85,B 0,C 180,E1 -25174.232,E2 -25174.232} C_VEL
LIN {X 0,Y 145.09,Z 436.846,A -85,B 0,C 180,E1 -25176.825,E2 -25176.825} C_VEL
LIN {X 0,Y 144.069,Z 435.219,A -85,B 0,C 180,E1 -25178.016,E2 -25178.016} C_VEL
LIN {X 0,Y 141.504,Z 432.711,A -85,B 0,C 180,E1 -25181.168,E2 -25181.168} C_VEL
LIN {X 0,Y 139.991,Z 429.904,A -85,B 0,C 180,E1 -25183.599,E2 -25183.599} C_VEL
LIN {X 0,Y 137.276,Z 427.875,A -85,B 0,C 180,E1 -25188.638,E2 -25188.638} C_VEL
LIN {X 0,Y 135.653,Z 424.788,A -85,B 0,C 180,E1 -25194.427,E2 -25194.427} C_VEL
LIN {X 0,Y 135.18,Z 423.782,A -85,B 0,C 180,E1 -25200.002,E2 -25200.002} C_VEL
LIN {X 0,Y 135.656,Z 424.796,A -85,B 0,C 180,E1 -25205.203,E2 -25205.203} C_VEL
LIN {X 0,Y 138.904,Z 429.349,A -85,B 0,C 180,E1 -25214.281,E2 -25214.281} C_VEL
LIN {X 0,Y 140.213,Z 430.212,A -85,B 0,C 180,E1 -25216.378,E2 -25216.378} C_VEL
LIN {X 0,Y 142.013,Z 433.352,A -85,B 0,C 180,E1 -25219.141,E2 -25219.141} C_VEL
LIN {X 0,Y 144.474,Z 435.737,A -85,B 0,C 180,E1 -25222.062,E2 -25222.062} C_VEL
LIN {X 0,Y 146.819,Z 439.134,A -85,B 0,C 180,E1 -25224.593,E2 -25224.593} C_VEL
LIN {X 0,Y 148.315,Z 440.715,A -85,B 0,C 180,E1 -25225.987,E2 -25225.987} C_VEL
LIN {X 0,Y 151.1,Z 444.522,A -85,B 0,C 180,E1 -25228.431,E2 -25228.431} C_VEL
LIN {X 0,Y 155.266,Z 450.563,A -85,B 0,C 180,E1 -25231.655,E2 -25231.655} C_VEL
LIN {X 0,Y 157.911,Z 455.184,A -85,B 0,C 180,E1 -25233.54,E2 -25233.54} C_VEL
LIN {X 0,Y 161.854,Z 463.318,A -85,B 0,C 180,E1 -25236.177,E2 -25236.177} C_VEL
LIN {X 0,Y 166.699,Z 474.578,A -85,B 0,C 180,E1 -25239.137,E2 -25239.137} C_VEL
LIN {X 0,Y 170.351,Z 484.757,A -85,B 0,C 180,E1 -25241.253,E2 -25241.253} C_VEL
LIN {X 0,Y 167.816,Z 519.505,A -85,B 0,C 180,E1 -25242.571,E2 -25242.571} C_VEL
LIN {X 0,Y 166.266,Z 530.498,A -85,B 0,C 180,E1 -25243.225,E2 -25243.225} C_VEL
LIN {X 0,Y 164.039,Z 541.383,A -85,B 0,C 180,E1 -25244.143,E2 -25244.143} C_VEL
LIN {X 0,Y 160.621,Z 553.825,A -85,B 0,C 180,E1 -25245.568,E2 -25245.568} C_VEL
LIN {X 0,Y 156.303,Z 566.084,A -85,B 0,C 180,E1 -25247.59,E2 -25247.59} C_VEL
LIN {X 0,Y 152.727,Z 574.806,A -85,B 0,C 180,E1 -25249.461,E2 -25249.461} C_VEL
LIN {X 0,Y 149.299,Z 582.221,A -85,B 0,C 180,E1 -25251.413,E2 -25251.413} C_VEL
LIN {X 0,Y 144.782,Z 591.012,A -85,B 0,C 180,E1 -25254.375,E2 -25254.375} C_VEL
LIN {X 0,Y 141.494,Z 597,A -85,B 0,C 180,E1 -25256.883,E2 -25256.883} C_VEL
LIN {X 0,Y 137.932,Z 603.35,A -85,B 0,C 180,E1 -25260.241,E2 -25260.241} C_VEL
LIN {X 0,Y 134.727,Z 608.587,A -85,B 0,C 180,E1 -25263.68,E2 -25263.68} C_VEL
LIN {X 0,Y 131.493,Z 613.681,A -85,B 0,C 180,E1 -25268.03,E2 -25268.03} C_VEL
LIN {X 0,Y 129.049,Z 617.649,A -85,B 0,C 180,E1 -25272.572,E2 -25272.572} C_VEL
LIN {X 0,Y 127.466,Z 620.592,A -85,B 0,C 180,E1 -25277.26,E2 -25277.26} C_VEL
LIN {X 0,Y 126.795,Z 622.099,A -85,B 0,C 180,E1 -25280.429,E2 -25280.429} C_VEL
LIN {X 0,Y 126.317,Z 623.636,A -85,B 0,C 180,E1 -25286.812,E2 -25286.812} C_VEL
LIN {X 0,Y 126.431,Z 623.921,A -85,B 0,C 180,E1 -25290.001,E2 -25290.001} C_VEL
LIN {X 0,Y 126.409,Z 623.033,A -85,B 0,C 180,E1 -25296.385,E2 -25296.385} C_VEL
LIN {X 0,Y 126.788,Z 622.098,A -85,B 0,C 180,E1 -25299.573,E2 -25299.573} C_VEL
LIN {X 0,Y 128.446,Z 618.739,A -85,B 0,C 180,E1 -25305.878,E2 -25305.878} C_VEL
LIN {X 0,Y 130.575,Z 615.107,A -85,B 0,C 180,E1 -25310.479,E2 -25310.479} C_VEL
LIN {X 0,Y 133.546,Z 610.374,A -85,B 0,C 180,E1 -25314.899,E2 -25314.899} C_VEL
LIN {X 0,Y 137.315,Z 604.405,A -85,B 0,C 180,E1 -25319.093,E2 -25319.093} C_VEL
LIN {X 0,Y 140.803,Z 598.312,A -85,B 0,C 180,E1 -25322.45,E2 -25322.45} C_VEL
LIN {X 0,Y 143.961,Z 592.569,A -85,B 0,C 180,E1 -25325.004,E2 -25325.004} C_VEL
LIN {X 0,Y 147.493,Z 585.917,A -85,B 0,C 180,E1 -25327.412,E2 -25327.412} C_VEL
LIN {X 0,Y 151.233,Z 578.093,A -85,B 0,C 180,E1 -25329.716,E2 -25329.716} C_VEL
LIN {X 0,Y 154.757,Z 570.015,A -85,B 0,C 180,E1 -25331.619,E2 -25331.619} C_VEL
LIN {X 0,Y 158.432,Z 560.258,A -85,B 0,C 180,E1 -25333.439,E2 -25333.439} C_VEL
LIN {X 0,Y 161.164,Z 551.872,A -85,B 0,C 180,E1 -25334.683,E2 -25334.683} C_VEL
LIN {X 0,Y 164.025,Z 541.371,A -85,B 0,C 180,E1 -25335.864,E2 -25335.864} C_VEL
LIN {X 0,Y 166.205,Z 531.208,A -85,B 0,C 180,E1 -25336.706,E2 -25336.706} C_VEL
LIN {X 0,Y 167.769,Z 520.156,A -85,B 0,C 180,E1 -25337.381,E2 -25337.381} C_VEL
LIN {X 0,Y 169.808,Z 493.931,A -85,B 0,C 180,E1 -25338.382,E2 -25338.382} C_VEL
LIN {X 0,Y 170.1,Z 489.75,A -85,B 0,C 180,E1 -25338.532,E2 -25338.532} C_VEL
LIN {X 0,Y 169.742,Z 486.784,A -85,B 0,C 180,E1 -25338.854,E2 -25338.854} C_VEL
LIN {X 0,Y 168.637,Z 484.29,A -85,B 0,C 180,E1 -25339.441,E2 -25339.441} C_VEL
LIN {X 0,Y 166.818,Z 481.892,A -85,B 0,C 180,E1 -25340.329,E2 -25340.329} C_VEL
LIN {X 0,Y 162.3,Z 476.933,A -85,B 0,C 180,E1 -25342.631,E2 -25342.631} C_VEL
LIN {X 0,Y 161.474,Z 475.488,A -85,B 0,C 180,E1 -25343.117,E2 -25343.117} C_VEL
LIN {X 0,Y 156.394,Z 463.751,A -85,B 0,C 180,E1 -25346.598,E2 -25346.598} C_VEL
LIN {X 0,Y 152.79,Z 456.722,A -85,B 0,C 180,E1 -25349.315,E2 -25349.315} C_VEL
LIN {X 0,Y 148.639,Z 450.512,A -85,B 0,C 180,E1 -25352.737,E2 -25352.737} C_VEL
LIN {X 0,Y 145.6,Z 446.278,A -85,B 0,C 180,E1 -25355.624,E2 -25355.624} C_VEL
LIN {X 0,Y 142.738,Z 442.406,A -85,B 0,C 180,E1 -25358.787,E2 -25358.787} C_VEL
LIN {X 0,Y 139.307,Z 438.189,A -85,B 0,C 180,E1 -25363.462,E2 -25363.462} C_VEL
LIN {X 0,Y 138.597,Z 436.711,A -85,B 0,C 180,E1 -25364.747,E2 -25364.747} C_VEL
LIN {X 0,Y 136.2,Z 434.718,A -85,B 0,C 180,E1 -25369.502,E2 -25369.502} C_VEL
LIN {X 0,Y 134.666,Z 431.625,A -85,B 0,C 180,E1 -25375.508,E2 -25375.508} C_VEL
LIN {X 0,Y 134.31,Z 430.863,A -85,B 0,C 180,E1 -25379.998,E2 -25379.998} C_VEL
LIN {X 0,Y 134.749,Z 431.853,A -85,B 0,C 180,E1 -25385.423,E2 -25385.423} C_VEL
LIN {X 0,Y 137.517,Z 436.104,A -85,B 0,C 180,E1 -25393.785,E2 -25393.785} C_VEL
LIN {X 0,Y 138.788,Z 437.031,A -85,B 0,C 180,E1 -25395.981,E2 -25395.981} C_VEL
LIN {X 0,Y 140.756,Z 440.372,A -85,B 0,C 180,E1 -25399.125,E2 -25399.125} C_VEL
LIN {X 0,Y 142.735,Z 442.368,A -85,B 0,C 180,E1 -25401.591,E2 -25401.591} C_VEL
LIN {X 0,Y 145.295,Z 446,A -85,B 0,C 180,E1 -25404.466,E2 -25404.466} C_VEL
LIN {X 0,Y 146.428,Z 447.423,A -85,B 0,C 180,E1 -25405.591,E2 -25405.591} C_VEL
LIN {X 0,Y 149.781,Z 452.241,A -85,B 0,C 180,E1 -25408.65,E2 -25408.65} C_VEL
LIN {X 0,Y 153.594,Z 457.94,A -85,B 0,C 180,E1 -25411.676,E2 -25411.676} C_VEL
LIN {X 0,Y 158.501,Z 466.1,A -85,B 0,C 180,E1 -25415.101,E2 -25415.101} C_VEL
LIN {X 0,Y 163.482,Z 475.292,A -85,B 0,C 180,E1 -25418.177,E2 -25418.177} C_VEL
LIN {X 0,Y 167.735,Z 484.435,A -85,B 0,C 180,E1 -25420.596,E2 -25420.596} C_VEL
LIN {X 0,Y 172.592,Z 496.739,A -85,B 0,C 180,E1 -25423.196,E2 -25423.196} C_VEL
LIN {X 0,Y 178.538,Z 511.757,A -85,B 0,C 180,E1 -25426.123,E2 -25426.123} C_VEL
LIN {X 0,Y 182.932,Z 521.614,A -85,B 0,C 180,E1 -25428.309,E2 -25428.309} C_VEL
LIN {X 0,Y 187.788,Z 531.449,A -85,B 0,C 180,E1 -25430.794,E2 -25430.794} C_VEL
LIN {X 0,Y 192.769,Z 540.483,A -85,B 0,C 180,E1 -25433.327,E2 -25433.327} C_VEL
LIN {X 0,Y 198.768,Z 549.596,A -85,B 0,C 180,E1 -25436.19,E2 -25436.19} C_VEL
LIN {X 0,Y 206.083,Z 559.016,A -85,B 0,C 180,E1 -25439.435,E2 -25439.435} C_VEL
LIN {X 0,Y 214.131,Z 567.539,A -85,B 0,C 180,E1 -25442.645,E2 -25442.645} C_VEL
LIN {X 0,Y 223.335,Z 575.354,A -85,B 0,C 180,E1 -25445.862,E2 -25445.862} C_VEL
LIN {X 0,Y 233.474,Z 582.206,A -85,B 0,C 180,E1 -25448.929,E2 -25448.929} C_VEL
LIN {X 0,Y 246.819,Z 589.725,A -85,B 0,C 180,E1 -25452.529,E2 -25452.529} C_VEL
LIN {X 0,Y 258.836,Z 595.701,A -85,B 0,C 180,E1 -25455.577,E2 -25455.577} C_VEL
LIN {X 0,Y 266.303,Z 599.365,A -85,B 0,C 180,E1 -25457.541,E2 -25457.541} C_VEL
LIN {X 0,Y 273.511,Z 602.984,A -85,B 0,C 180,E1 -25459.638,E2 -25459.638} C_VEL
LIN {X 0,Y 278.7,Z 605.574,A -85,B 0,C 180,E1 -25461.297,E2 -25461.297} C_VEL
LIN {X 0,Y 283.095,Z 608.166,A -85,B 0,C 180,E1 -25463.221,E2 -25463.221} C_VEL
LIN {X 0,Y 285.315,Z 609.432,A -85,B 0,C 180,E1 -25464.345,E2 -25464.345} C_VEL
LIN {X 0,Y 288.728,Z 611.18,A -85,B 0,C 180,E1 -25466.352,E2 -25466.352} C_VEL
LIN {X 0,Y 289.859,Z 611.662,A -85,B 0,C 180,E1 -25467.22,E2 -25467.22} C_VEL
LIN {X 0,Y 291.121,Z 612.168,A -85,B 0,C 180,E1 -25468.616,E2 -25468.616} C_VEL
LIN {X 0,Y 291.781,Z 612.314,A -85,B 0,C 180,E1 -25470,E2 -25470} C_VEL
LIN {X 0,Y 291.141,Z 612.17,A -85,B 0,C 180,E1 -25471.383,E2 -25471.383} C_VEL
LIN {X 0,Y 289.86,Z 611.663,A -85,B 0,C 180,E1 -25472.779,E2 -25472.779} C_VEL
LIN {X 0,Y 287.818,Z 610.75,A -85,B 0,C 180,E1 -25474.2,E2 -25474.2} C_VEL
LIN {X 0,Y 285.278,Z 609.434,A -85,B 0,C 180,E1 -25475.655,E2 -25475.655} C_VEL
LIN {X 0,Y 282.29,Z 607.727,A -85,B 0,C 180,E1 -25477.15,E2 -25477.15} C_VEL
LIN {X 0,Y 278.712,Z 605.575,A -85,B 0,C 180,E1 -25478.701,E2 -25478.701} C_VEL
LIN {X 0,Y 271.913,Z 602.199,A -85,B 0,C 180,E1 -25480.842,E2 -25480.842} C_VEL
LIN {X 0,Y 263.496,Z 597.97,A -85,B 0,C 180,E1 -25483.217,E2 -25483.217} C_VEL
LIN {X 0,Y 251.815,Z 592.263,A -85,B 0,C 180,E1 -25486.205,E2 -25486.205} C_VEL
LIN {X 0,Y 238.733,Z 585.371,A -85,B 0,C 180,E1 -25489.606,E2 -25489.606} C_VEL
LIN {X 0,Y 225.825,Z 577.147,A -85,B 0,C 180,E1 -25493.356,E2 -25493.356} C_VEL
LIN {X 0,Y 216.17,Z 569.383,A -85,B 0,C 180,E1 -25496.616,E2 -25496.616} C_VEL
LIN {X 0,Y 208.272,Z 561.456,A -85,B 0,C 180,E1 -25499.67,E2 -25499.67} C_VEL
LIN {X 0,Y 200.819,Z 552.408,A -85,B 0,C 180,E1 -25502.871,E2 -25502.871} C_VEL
LIN {X 0,Y 194.744,Z 543.662,A -85,B 0,C 180,E1 -25505.71,E2 -25505.71} C_VEL
LIN {X 0,Y 189.759,Z 535.223,A -85,B 0,C 180,E1 -25508.202,E2 -25508.202} C_VEL
LIN {X 0,Y 184.011,Z 523.953,A -85,B 0,C 180,E1 -25511.14,E2 -25511.14} C_VEL
LIN {X 0,Y 178.702,Z 512.129,A -85,B 0,C 180,E1 -25513.83,E2 -25513.83} C_VEL
LIN {X 0,Y 170.666,Z 491.561,A -85,B 0,C 180,E1 -25517.82,E2 -25517.82} C_VEL
LIN {X 0,Y 165.537,Z 479.47,A -85,B 0,C 180,E1 -25520.639,E2 -25520.639} C_VEL
LIN {X 0,Y 160.82,Z 470.233,A -85,B 0,C 180,E1 -25523.426,E2 -25523.426} C_VEL
LIN {X 0,Y 155.677,Z 461.294,A -85,B 0,C 180,E1 -25526.814,E2 -25526.814} C_VEL
LIN {X 0,Y 151.068,Z 454.143,A -85,B 0,C 180,E1 -25530.282,E2 -25530.282} C_VEL
LIN {X 0,Y 148.44,Z 450.296,A -85,B 0,C 180,E1 -25532.521,E2 -25532.521} C_VEL
LIN {X 0,Y 145.622,Z 446.319,A -85,B 0,C 180,E1 -25535.213,E2 -25535.213} C_VEL
LIN {X 0,Y 142.923,Z 442.725,A -85,B 0,C 180,E1 -25538.171,E2 -25538.171} C_VEL
LIN {X 0,Y 142.237,Z 441.771,A -85,B 0,C 180,E1 -25539.01,E2 -25539.01} C_VEL
LIN {X 0,Y 139.696,Z 438.902,A -85,B 0,C 180,E1 -25542.433,E2 -25542.433} C_VEL
LIN {X 0,Y 138.696,Z 436.804,A -85,B 0,C 180,E1 -25544.197,E2 -25544.197} C_VEL
LIN {X 0,Y 136.165,Z 434.759,A -85,B 0,C 180,E1 -25549.183,E2 -25549.183} C_VEL
LIN {X 0,Y 134.657,Z 431.675,A -85,B 0,C 180,E1 -25555.136,E2 -25555.136} C_VEL
LIN {X 0,Y 134.313,Z 430.838,A -85,B 0,C 180,E1 -25560.002,E2 -25560.002} C_VEL
LIN {X 0,Y 134.719,Z 431.797,A -85,B 0,C 180,E1 -25564.865,E2 -25564.865} C_VEL
LIN {X 0,Y 137.656,Z 436.215,A -85,B 0,C 180,E1 -25573.66,E2 -25573.66} C_VEL
LIN {X 0,Y 138.75,Z 436.915,A -85,B 0,C 180,E1 -25575.518,E2 -25575.518} C_VEL
LIN {X 0,Y 140.582,Z 440.12,A -85,B 0,C 180,E1 -25578.492,E2 -25578.492} C_VEL
LIN {X 0,Y 142.646,Z 442.21,A -85,B 0,C 180,E1 -25581.091,E2 -25581.091} C_VEL
LIN {X 0,Y 145.066,Z 445.714,A -85,B 0,C 180,E1 -25583.844,E2 -25583.844} C_VEL
LIN {X 0,Y 146.518,Z 447.545,A -85,B 0,C 180,E1 -25585.292,E2 -25585.292} C_VEL
LIN {X 0,Y 149.788,Z 452.259,A -85,B 0,C 180,E1 -25588.27,E2 -25588.27} C_VEL
LIN {X 0,Y 153.279,Z 457.461,A -85,B 0,C 180,E1 -25591.054,E2 -25591.054} C_VEL
LIN {X 0,Y 156.988,Z 465.118,A -85,B 0,C 180,E1 -25593.836,E2 -25593.836} C_VEL
LIN {X 0,Y 162.201,Z 477.242,A -85,B 0,C 180,E1 -25597.346,E2 -25597.346} C_VEL
LIN {X 0,Y 165.633,Z 487.18,A -85,B 0,C 180,E1 -25599.53,E2 -25599.53} C_VEL
LIN {X 0,Y 163.09,Z 519.463,A -85,B 0,C 180,E1 -25600.745,E2 -25600.745} C_VEL
LIN {X 0,Y 161.433,Z 530.632,A -85,B 0,C 180,E1 -25601.413,E2 -25601.413} C_VEL
LIN {X 0,Y 158.877,Z 542.45,A -85,B 0,C 180,E1 -25602.425,E2 -25602.425} C_VEL
LIN {X 0,Y 155.067,Z 555.304,A -85,B 0,C 180,E1 -25603.989,E2 -25603.989} C_VEL
LIN {X 0,Y 151.139,Z 565.889,A -85,B 0,C 180,E1 -25605.775,E2 -25605.775} C_VEL
LIN {X 0,Y 147.394,Z 574.61,A -85,B 0,C 180,E1 -25607.664,E2 -25607.664} C_VEL
LIN {X 0,Y 143.806,Z 582.026,A -85,B 0,C 180,E1 -25609.645,E2 -25609.645} C_VEL
LIN {X 0,Y 139.046,Z 590.816,A -85,B 0,C 180,E1 -25612.662,E2 -25612.662} C_VEL
LIN {X 0,Y 135.573,Z 596.804,A -85,B 0,C 180,E1 -25615.235,E2 -25615.235} C_VEL
LIN {X 0,Y 131.461,Z 603.654,A -85,B 0,C 180,E1 -25619.025,E2 -25619.025} C_VEL
LIN {X 0,Y 128.392,Z 608.392,A -85,B 0,C 180,E1 -25622.273,E2 -25622.273} C_VEL
LIN {X 0,Y 124.917,Z 613.485,A -85,B 0,C 180,E1 -25626.808,E2 -25626.808} C_VEL
LIN {X 0,Y 122.246,Z 617.452,A -85,B 0,C 180,E1 -25631.568,E2 -25631.568} C_VEL
LIN {X 0,Y 120.525,Z 620.396,A -85,B 0,C 180,E1 -25636.513,E2 -25636.513} C_VEL
LIN {X 0,Y 119.787,Z 621.903,A -85,B 0,C 180,E1 -25639.864,E2 -25639.864} C_VEL
LIN {X 0,Y 119.231,Z 623.441,A -85,B 0,C 180,E1 -25646.622,E2 -25646.622} C_VEL
LIN {X 0,Y 119.337,Z 623.726,A -85,B 0,C 180,E1 -25650.001,E2 -25650.001} C_VEL
LIN {X 0,Y 119.332,Z 622.837,A -85,B 0,C 180,E1 -25656.765,E2 -25656.765} C_VEL
LIN {X 0,Y 119.759,Z 621.902,A -85,B 0,C 180,E1 -25660.141,E2 -25660.141} C_VEL
LIN {X 0,Y 121.584,Z 618.543,A -85,B 0,C 180,E1 -25666.8,E2 -25666.8} C_VEL
LIN {X 0,Y 123.928,Z 614.912,A -85,B 0,C 180,E1 -25671.631,E2 -25671.631} C_VEL
LIN {X 0,Y 127.11,Z 610.178,A -85,B 0,C 180,E1 -25676.253,E2 -25676.253} C_VEL
LIN {X 0,Y 130.612,Z 605.019,A -85,B 0,C 180,E1 -25680.08,E2 -25680.08} C_VEL
LIN {X 0,Y 134.048,Z 599.427,A -85,B 0,C 180,E1 -25683.402,E2 -25683.402} C_VEL
LIN {X 0,Y 137.319,Z 593.934,A -85,B 0,C 180,E1 -25686.056,E2 -25686.056} C_VEL
LIN {X 0,Y 141.894,Z 585.721,A -85,B 0,C 180,E1 -25689.162,E2 -25689.162} C_VEL
LIN {X 0,Y 145.843,Z 577.898,A -85,B 0,C 180,E1 -25691.499,E2 -25691.499} C_VEL
LIN {X 0,Y 149.517,Z 569.819,A -85,B 0,C 180,E1 -25693.428,E2 -25693.428} C_VEL
LIN {X 0,Y 153.338,Z 560.063,A -85,B 0,C 180,E1 -25695.269,E2 -25695.269} C_VEL
LIN {X 0,Y 156.202,Z 551.677,A -85,B 0,C 180,E1 -25696.512,E2 -25696.512} C_VEL
LIN {X 0,Y 159.168,Z 541.176,A -85,B 0,C 180,E1 -25697.697,E2 -25697.697} C_VEL
LIN {X 0,Y 161.496,Z 530.625,A -85,B 0,C 180,E1 -25698.563,E2 -25698.563} C_VEL
LIN {X 0,Y 163.019,Z 520.22,A -85,B 0,C 180,E1 -25699.205,E2 -25699.205} C_VEL
LIN {X 0,Y 164.902,Z 497.341,A -85,B 0,C 180,E1 -25700.099,E2 -25700.099} C_VEL
LIN {X 0,Y 165.635,Z 487.168,A -85,B 0,C 180,E1 -25700.47,E2 -25700.47} C_VEL
LIN {X 0,Y 161.474,Z 475.488,A -85,B 0,C 180,E1 -25703.117,E2 -25703.117} C_VEL
LIN {X 0,Y 159.163,Z 471.698,A -85,B 0,C 180,E1 -25704.519,E2 -25704.519} C_VEL
LIN {X 0,Y 154.751,Z 466.924,A -85,B 0,C 180,E1 -25707.259,E2 -25707.259} C_VEL
LIN {X 0,Y 151.26,Z 463.549,A -85,B 0,C 180,E1 -25709.668,E2 -25709.668} C_VEL
LIN {X 0,Y 148.259,Z 459.621,A -85,B 0,C 180,E1 -25712.09,E2 -25712.09} C_VEL
LIN {X 0,Y 145.701,Z 455.768,A -85,B 0,C 180,E1 -25714.46,E2 -25714.46} C_VEL
LIN {X 0,Y 143.501,Z 452.547,A -85,B 0,C 180,E1 -25716.741,E2 -25716.741} C_VEL
LIN {X 0,Y 140.574,Z 448.323,A -85,B 0,C 180,E1 -25720.276,E2 -25720.276} C_VEL
LIN {X 0,Y 138.065,Z 445.271,A -85,B 0,C 180,E1 -25723.93,E2 -25723.93} C_VEL
LIN {X 0,Y 137.214,Z 443.56,A -85,B 0,C 180,E1 -25725.539,E2 -25725.539} C_VEL
LIN {X 0,Y 134.552,Z 440.795,A -85,B 0,C 180,E1 -25731.74,E2 -25731.74} C_VEL
LIN {X 0,Y 133.688,Z 438.524,A -85,B 0,C 180,E1 -25736.231,E2 -25736.231} C_VEL
LIN {X 0,Y 133.446,Z 437.905,A -85,B 0,C 180,E1 -25739.998,E2 -25739.998} C_VEL
LIN {X 0,Y 133.787,Z 438.788,A -85,B 0,C 180,E1 -25744.895,E2 -25744.895} C_VEL
LIN {X 0,Y 136.421,Z 443.059,A -85,B 0,C 180,E1 -25753.403,E2 -25753.403} C_VEL
LIN {X 0,Y 137.399,Z 443.845,A -85,B 0,C 180,E1 -25755.196,E2 -25755.196} C_VEL
LIN {X 0,Y 139.816,Z 447.694,A -85,B 0,C 180,E1 -25759.138,E2 -25759.138} C_VEL
LIN {X 0,Y 141.05,Z 449.005,A -85,B 0,C 180,E1 -25760.734,E2 -25760.734} C_VEL
LIN {X 0,Y 143.81,Z 452.869,A -85,B 0,C 180,E1 -25763.967,E2 -25763.967} C_VEL
LIN {X 0,Y 147.431,Z 458.334,A -85,B 0,C 180,E1 -25767.555,E2 -25767.555} C_VEL
LIN {X 0,Y 151.408,Z 464.512,A -85,B 0,C 180,E1 -25770.901,E2 -25770.901} C_VEL
LIN {X 0,Y 156.922,Z 474.316,A -85,B 0,C 180,E1 -25774.918,E2 -25774.918} C_VEL
LIN {X 0,Y 161.421,Z 483.362,A -85,B 0,C 180,E1 -25777.81,E2 -25777.81} C_VEL
LIN {X 0,Y 165.359,Z 492.849,A -85,B 0,C 180,E1 -25780.179,E2 -25780.179} C_VEL
LIN {X 0,Y 172.693,Z 512.648,A -85,B 0,C 180,E1 -25784.281,E2 -25784.281} C_VEL
LIN {X 0,Y 176.114,Z 521.162,A -85,B 0,C 180,E1 -25786.222,E2 -25786.222} C_VEL
LIN {X 0,Y 180.13,Z 530.48,A -85,B 0,C 180,E1 -25788.595,E2 -25788.595} C_VEL
LIN {X 0,Y 184.888,Z 540.217,A -85,B 0,C 180,E1 -25791.392,E2 -25791.392} C_VEL
LIN {X 0,Y 190.233,Z 549.459,A -85,B 0,C 180,E1 -25794.366,E2 -25794.366} C_VEL
LIN {X 0,Y 196.518,Z 558.392,A -85,B 0,C 180,E1 -25797.558,E2 -25797.558} C_VEL
LIN {X 0,Y 204.517,Z 567.829,A -85,B 0,C 180,E1 -25801.243,E2 -25801.243} C_VEL
LIN {X 0,Y 212.936,Z 575.622,A -85,B 0,C 180,E1 -25804.591,E2 -25804.591} C_VEL
LIN {X 0,Y 221.824,Z 582.195,A -85,B 0,C 180,E1 -25807.654,E2 -25807.654} C_VEL
LIN {X 0,Y 233.839,Z 589.202,A -85,B 0,C 180,E1 -25811.211,E2 -25811.211} C_VEL
LIN {X 0,Y 247.542,Z 595.904,A -85,B 0,C 180,E1 -25814.857,E2 -25814.857} C_VEL
LIN {X 0,Y 257.26,Z 600.229,A -85,B 0,C 180,E1 -25817.376,E2 -25817.376} C_VEL
LIN {X 0,Y 264.511,Z 603.544,A -85,B 0,C 180,E1 -25819.44,E2 -25819.44} C_VEL
LIN {X 0,Y 270.245,Z 606.095,A -85,B 0,C 180,E1 -25821.193,E2 -25821.193} C_VEL
LIN {X 0,Y 274.123,Z 607.952,A -85,B 0,C 180,E1 -25822.635,E2 -25822.635} C_VEL
LIN {X 0,Y 277.398,Z 609.649,A -85,B 0,C 180,E1 -25824.183,E2 -25824.183} C_VEL
LIN {X 0,Y 281.621,Z 611.565,A -85,B 0,C 180,E1 -25826.565,E2 -25826.565} C_VEL
LIN {X 0,Y 282.437,Z 611.883,A -85,B 0,C 180,E1 -25827.147,E2 -25827.147} C_VEL
LIN {X 0,Y 283.887,Z 612.444,A -85,B 0,C 180,E1 -25828.581,E2 -25828.581} C_VEL
LIN {X 0,Y 284.65,Z 612.628,A -85,B 0,C 180,E1 -25830,E2 -25830} C_VEL
LIN {X 0,Y 283.902,Z 612.444,A -85,B 0,C 180,E1 -25831.418,E2 -25831.418} C_VEL
LIN {X 0,Y 282.437,Z 611.884,A -85,B 0,C 180,E1 -25832.852,E2 -25832.852} C_VEL
LIN {X 0,Y 280.131,Z 610.963,A -85,B 0,C 180,E1 -25834.316,E2 -25834.316} C_VEL
LIN {X 0,Y 275.895,Z 608.874,A -85,B 0,C 180,E1 -25836.563,E2 -25836.563} C_VEL
LIN {X 0,Y 274.165,Z 607.952,A -85,B 0,C 180,E1 -25837.363,E2 -25837.363} C_VEL
LIN {X 0,Y 269.629,Z 605.828,A -85,B 0,C 180,E1 -25838.997,E2 -25838.997} C_VEL
LIN {X 0,Y 261.371,Z 602.13,A -85,B 0,C 180,E1 -25841.476,E2 -25841.476} C_VEL
LIN {X 0,Y 253.163,Z 598.45,A -85,B 0,C 180,E1 -25843.685,E2 -25843.685} C_VEL
LIN {X 0,Y 240.454,Z 592.59,A -85,B 0,C 180,E1 -25846.994,E2 -25846.994} C_VEL
LIN {X 0,Y 228.731,Z 586.484,A -85,B 0,C 180,E1 -25850.227,E2 -25850.227} C_VEL
LIN {X 0,Y 215.958,Z 578.008,A -85,B 0,C 180,E1 -25854.329,E2 -25854.329} C_VEL
LIN {X 0,Y 206.664,Z 570.032,A -85,B 0,C 180,E1 -25857.852,E2 -25857.852} C_VEL
LIN {X 0,Y 199.672,Z 562.406,A -85,B 0,C 180,E1 -25860.93,E2 -25860.93} C_VEL
LIN {X 0,Y 192.581,Z 553.026,A -85,B 0,C 180,E1 -25864.397,E2 -25864.397} C_VEL
LIN {X 0,Y 187.442,Z 544.9,A -85,B 0,C 180,E1 -25867.158,E2 -25867.158} C_VEL
LIN {X 0,Y 182.004,Z 534.408,A -85,B 0,C 180,E1 -25870.306,E2 -25870.306} C_VEL
LIN {X 0,Y 177.683,Z 524.895,A -85,B 0,C 180,E1 -25872.866,E2 -25872.866} C_VEL
LIN {X 0,Y 173.073,Z 513.651,A -85,B 0,C 180,E1 -25875.537,E2 -25875.537} C_VEL
LIN {X 0,Y 164.818,Z 491.43,A -85,B 0,C 180,E1 -25880.141,E2 -25880.141} C_VEL
LIN {X 0,Y 161.019,Z 482.536,A -85,B 0,C 180,E1 -25882.436,E2 -25882.436} C_VEL
LIN {X 0,Y 157.023,Z 474.557,A -85,B 0,C 180,E1 -25885.01,E2 -25885.01} C_VEL
LIN {X 0,Y 152.567,Z 466.54,A -85,B 0,C 180,E1 -25888.195,E2 -25888.195} C_VEL
LIN {X 0,Y 148.171,Z 459.445,A -85,B 0,C 180,E1 -25891.785,E2 -25891.785} C_VEL
LIN {X 0,Y 145.634,Z 455.712,A -85,B 0,C 180,E1 -25894.134,E2 -25894.134} C_VEL
LIN {X 0,Y 143.496,Z 452.53,A -85,B 0,C 180,E1 -25896.361,E2 -25896.361} C_VEL
LIN {X 0,Y 140.908,Z 448.729,A -85,B 0,C 180,E1 -25899.459,E2 -25899.459} C_VEL
LIN {X 0,Y 138.06,Z 445.258,A -85,B 0,C 180,E1 -25903.553,E2 -25903.553} C_VEL
LIN {X 0,Y 137.21,Z 443.544,A -85,B 0,C 180,E1 -25905.163,E2 -25905.163} C_VEL
LIN {X 0,Y 134.908,Z 441.377,A -85,B 0,C 180,E1 -25910.206,E2 -25910.206} C_VEL
LIN {X 0,Y 133.684,Z 438.544,A -85,B 0,C 180,E1 -25915.856,E2 -25915.856} C_VEL
LIN {X 0,Y 133.447,Z 437.892,A -85,B 0,C 180,E1 -25920.002,E2 -25920.002} C_VEL
LIN {X 0,Y 133.786,Z 438.812,A -85,B 0,C 180,E1 -25924.521,E2 -25924.521} C_VEL
LIN {X 0,Y 136.343,Z 443.008,A -85,B 0,C 180,E1 -25932.863,E2 -25932.863} C_VEL
LIN {X 0,Y 137.451,Z 443.942,A -85,B 0,C 180,E1 -25934.909,E2 -25934.909} C_VEL
LIN {X 0,Y 139.531,Z 447.335,A -85,B 0,C 180,E1 -25938.351,E2 -25938.351} C_VEL
LIN {X 0,Y 141.092,Z 449.111,A -85,B 0,C 180,E1 -25940.408,E2 -25940.408} C_VEL
LIN {X 0,Y 144.583,Z 454.064,A -85,B 0,C 180,E1 -25944.406,E2 -25944.406} C_VEL
LIN {X 0,Y 147.649,Z 458.66,A -85,B 0,C 180,E1 -25947.365,E2 -25947.365} C_VEL
LIN {X 0,Y 150.577,Z 463.301,A -85,B 0,C 180,E1 -25949.865,E2 -25949.865} C_VEL
LIN {X 0,Y 153.8,Z 470.291,A -85,B 0,C 180,E1 -25952.476,E2 -25952.476} C_VEL
LIN {X 0,Y 158.467,Z 481.74,A -85,B 0,C 180,E1 -25955.893,E2 -25955.893} C_VEL
LIN {X 0,Y 161.01,Z 489.464,A -85,B 0,C 180,E1 -25957.67,E2 -25957.67} C_VEL
LIN {X 0,Y 158.549,Z 519.274,A -85,B 0,C 180,E1 -25958.801,E2 -25958.801} C_VEL
LIN {X 0,Y 156.85,Z 530.351,A -85,B 0,C 180,E1 -25959.465,E2 -25959.465} C_VEL
LIN {X 0,Y 154.49,Z 540.993,A -85,B 0,C 180,E1 -25960.363,E2 -25960.363} C_VEL
LIN {X 0,Y 150.818,Z 553.435,A -85,B 0,C 180,E1 -25961.792,E2 -25961.792} C_VEL
LIN {X 0,Y 146.137,Z 565.694,A -85,B 0,C 180,E1 -25963.834,E2 -25963.834} C_VEL
LIN {X 0,Y 142.222,Z 574.415,A -85,B 0,C 180,E1 -25965.735,E2 -25965.735} C_VEL
LIN {X 0,Y 138.452,Z 581.83,A -85,B 0,C 180,E1 -25967.735,E2 -25967.735} C_VEL
LIN {X 0,Y 133.46,Z 590.621,A -85,B 0,C 180,E1 -25970.81,E2 -25970.81} C_VEL
LIN {X 0,Y 129.787,Z 596.608,A -85,B 0,C 180,E1 -25973.442,E2 -25973.442} C_VEL
LIN {X 0,Y 125.663,Z 603.002,A -85,B 0,C 180,E1 -25977.028,E2 -25977.028} C_VEL
LIN {X 0,Y 122.144,Z 608.196,A -85,B 0,C 180,E1 -25980.721,E2 -25980.721} C_VEL
LIN {X 0,Y 118.408,Z 613.29,A -85,B 0,C 180,E1 -25985.452,E2 -25985.452} C_VEL
LIN {X 0,Y 115.497,Z 617.256,A -85,B 0,C 180,E1 -25990.449,E2 -25990.449} C_VEL
LIN {X 0,Y 113.616,Z 620.201,A -85,B 0,C 180,E1 -25995.676,E2 -25995.676} C_VEL
LIN {X 0,Y 112.779,Z 621.708,A -85,B 0,C 180,E1 -25999.226,E2 -25999.226} C_VEL
LIN {X 0,Y 112.139,Z 623.246,A -85,B 0,C 180,E1 -26006.408,E2 -26006.408} C_VEL
LIN {X 0,Y 112.253,Z 623.532,A -85,B 0,C 180,E1 -26010.001,E2 -26010.001} C_VEL
LIN {X 0,Y 112.267,Z 622.641,A -85,B 0,C 180,E1 -26017.193,E2 -26017.193} C_VEL
LIN {X 0,Y 112.757,Z 621.706,A -85,B 0,C 180,E1 -26020.778,E2 -26020.778} C_VEL
LIN {X 0,Y 114.757,Z 618.347,A -85,B 0,C 180,E1 -26027.832,E2 -26027.832} C_VEL
LIN {X 0,Y 117.342,Z 614.716,A -85,B 0,C 180,E1 -26032.912,E2 -26032.912} C_VEL
LIN {X 0,Y 120.761,Z 609.983,A -85,B 0,C 180,E1 -26037.748,E2 -26037.748} C_VEL
LIN {X 0,Y 124.975,Z 604.028,A -85,B 0,C 180,E1 -26042.279,E2 -26042.279} C_VEL
LIN {X 0,Y 128.978,Z 597.918,A -85,B 0,C 180,E1 -26045.858,E2 -26045.858} C_VEL
LIN {X 0,Y 132.545,Z 592.178,A -85,B 0,C 180,E1 -26048.538,E2 -26048.538} C_VEL
LIN {X 0,Y 136.445,Z 585.526,A -85,B 0,C 180,E1 -26051.051,E2 -26051.051} C_VEL
LIN {X 0,Y 140.587,Z 577.703,A -85,B 0,C 180,E1 -26053.423,E2 -26053.423} C_VEL
LIN {X 0,Y 144.433,Z 569.624,A -85,B 0,C 180,E1 -26055.369,E2 -26055.369} C_VEL
LIN {X 0,Y 148.431,Z 559.868,A -85,B 0,C 180,E1 -26057.215,E2 -26057.215} C_VEL
LIN {X 0,Y 151.409,Z 551.482,A -85,B 0,C 180,E1 -26058.459,E2 -26058.459} C_VEL
LIN {X 0,Y 154.484,Z 540.981,A -85,B 0,C 180,E1 -26059.642,E2 -26059.642} C_VEL
LIN {X 0,Y 156.909,Z 530.356,A -85,B 0,C 180,E1 -26060.509,E2 -26060.509} C_VEL
LIN {X 0,Y 158.446,Z 520.355,A -85,B 0,C 180,E1 -26061.129,E2 -26061.129} C_VEL
LIN {X 0,Y 160.446,Z 497.146,A -85,B 0,C 180,E1 -26062.041,E2 -26062.041} C_VEL
LIN {X 0,Y 161.017,Z 489.397,A -85,B 0,C 180,E1 -26062.332,E2 -26062.332} C_VEL
LIN {X 0,Y 157.571,Z 479.406,A -85,B 0,C 180,E1 -26064.736,E2 -26064.736} C_VEL
LIN {X 0,Y 152.947,Z 468.324,A -85,B 0,C 180,E1 -26068.196,E2 -26068.196} C_VEL
LIN {X 0,Y 149.762,Z 461.871,A -85,B 0,C 180,E1 -26070.815,E2 -26070.815} C_VEL
LIN {X 0,Y 148.259,Z 459.621,A -85,B 0,C 180,E1 -26072.09,E2 -26072.09} C_VEL
LIN {X 0,Y 146.864,Z 457.785,A -85,B 0,C 180,E1 -26073.32,E2 -26073.32} C_VEL
LIN {X 0,Y 145.349,Z 456.568,A -85,B 0,C 180,E1 -26074.66,E2 -26074.66} C_VEL
LIN {X 0,Y 142.279,Z 455.34,A -85,B 0,C 180,E1 -26077.541,E2 -26077.541} C_VEL
LIN {X 0,Y 138.24,Z 453.943,A -85,B 0,C 180,E1 -26082.196,E2 -26082.196} C_VEL
LIN {X 0,Y 137.213,Z 452.876,A -85,B 0,C 180,E1 -26083.757,E2 -26083.757} C_VEL
LIN {X 0,Y 135.768,Z 450.282,A -85,B 0,C 180,E1 -26086.528,E2 -26086.528} C_VEL
LIN {X 0,Y 133.297,Z 447.215,A -85,B 0,C 180,E1 -26093.185,E2 -26093.185} C_VEL
LIN {X 0,Y 132.733,Z 445.419,A -85,B 0,C 180,E1 -26096.963,E2 -26096.963} C_VEL
LIN {X 0,Y 132.579,Z 444.962,A -85,B 0,C 180,E1 -26099.998,E2 -26099.998} C_VEL
LIN {X 0,Y 132.859,Z 445.801,A -85,B 0,C 180,E1 -26104.549,E2 -26104.549} C_VEL
LIN {X 0,Y 135.208,Z 449.925,A -85,B 0,C 180,E1 -26112.761,E2 -26112.761} C_VEL
LIN {X 0,Y 136.103,Z 450.783,A -85,B 0,C 180,E1 -26114.531,E2 -26114.531} C_VEL
LIN {X 0,Y 138.485,Z 454.549,A -85,B 0,C 180,E1 -26118.599,E2 -26118.599} C_VEL
LIN {X 0,Y 139.523,Z 455.889,A -85,B 0,C 180,E1 -26120.039,E2 -26120.039} C_VEL
LIN {X 0,Y 142.533,Z 460.32,A -85,B 0,C 180,E1 -26123.712,E2 -26123.712} C_VEL
LIN {X 0,Y 145.582,Z 465.12,A -85,B 0,C 180,E1 -26126.854,E2 -26126.854} C_VEL
LIN {X 0,Y 149.387,Z 471.486,A -85,B 0,C 180,E1 -26130.232,E2 -26130.232} C_VEL
LIN {X 0,Y 153.892,Z 479.892,A -85,B 0,C 180,E1 -26133.72,E2 -26133.72} C_VEL
LIN {X 0,Y 158.044,Z 488.707,A -85,B 0,C 180,E1 -26136.594,E2 -26136.594} C_VEL
LIN {X 0,Y 161.953,Z 498.556,A -85,B 0,C 180,E1 -26139.116,E2 -26139.116} C_VEL
LIN {X 0,Y 167.933,Z 515.895,A -85,B 0,C 180,E1 -26142.847,E2 -26142.847} C_VEL
LIN {X 0,Y 172.593,Z 528.456,A -85,B 0,C 180,E1 -26145.98,E2 -26145.98} C_VEL
LIN {X 0,Y 176.951,Z 538.84,A -85,B 0,C 180,E1 -26148.991,E2 -26148.991} C_VEL
LIN {X 0,Y 181.982,Z 549.096,A -85,B 0,C 180,E1 -26152.34,E2 -26152.34} C_VEL
LIN {X 0,Y 187.922,Z 558.665,A -85,B 0,C 180,E1 -26155.876,E2 -26155.876} C_VEL
LIN {X 0,Y 195.269,Z 568.112,A -85,B 0,C 180,E1 -26159.743,E2 -26159.743} C_VEL
LIN {X 0,Y 202.931,Z 575.92,A -85,B 0,C 180,E1 -26163.242,E2 -26163.242} C_VEL
LIN {X 0,Y 211.115,Z 582.506,A -85,B 0,C 180,E1 -26166.454,E2 -26166.454} C_VEL
LIN {X 0,Y 220.974,Z 588.717,A -85,B 0,C 180,E1 -26169.751,E2 -26169.751} C_VEL
LIN {X 0,Y 234.391,Z 595.435,A -85,B 0,C 180,E1 -26173.632,E2 -26173.632} C_VEL
LIN {X 0,Y 246.351,Z 600.529,A -85,B 0,C 180,E1 -26176.807,E2 -26176.807} C_VEL
LIN {X 0,Y 253.918,Z 603.533,A -85,B 0,C 180,E1 -26178.828,E2 -26178.828} C_VEL
